LIN {X 0,Y 142.755,Z 442.404,A -85,B 0,C 180,E1 -25401.516,E2 -25401.516} C_VEL
LIN {X 0,Y 145.368,Z 446.098,A -85,B 0,C 180,E1 -25404.454,E2 -25404.454} C_VEL
LIN {X 0,Y 146.59,Z 447.682,A -85,B 0,C 180,E1 -25405.67,E2 -25405.67} C_VEL
LIN {X 0,Y 149.941,Z 452.496,A -85,B 0,C 180,E1 -25408.714,E2 -25408.714} C_VEL
LIN {X 0,Y 154.159,Z 458.757,A -85,B 0,C 180,E1 -25412.023,E2 -25412.023} C_VEL
LIN {X 0,Y 159.816,Z 468.413,A -85,B 0,C 180,E1 -25415.888,E2 -25415.888} C_VEL
LIN {X 0,Y 164.555,Z 477.501,A -85,B 0,C 180,E1 -25418.752,E2 -25418.752} C_VEL
LIN {X 0,Y 166.086,Z 481.604,A -85,B 0,C 180,E1 -25419.683,E2 -25419.683} C_VEL
LIN {X 0,Y 164.265,Z 506.272,A -85,B 0,C 180,E1 -25420.566,E2 -25420.566} C_VEL
LIN {X 0,Y 162.83,Z 520.798,A -85,B 0,C 180,E1 -25421.21,E2 -25421.21} C_VEL
LIN {X 0,Y 160.572,Z 533.522,A -85,B 0,C 180,E1 -25422.156,E2 -25422.156} C_VEL
LIN {X 0,Y 157.451,Z 545.977,A -85,B 0,C 180,E1 -25423.503,E2 -25423.503} C_VEL
LIN {X 0,Y 153.61,Z 557.923,A -85,B 0,C 180,E1 -25425.297,E2 -25425.297} C_VEL
LIN {X 0,Y 149.443,Z 568.566,A -85,B 0,C 180,E1 -25427.467,E2 -25427.467} C_VEL
LIN {X 0,Y 144.921,Z 578.272,A -85,B 0,C 180,E1 -25430.017,E2 -25430.017} C_VEL
LIN {X 0,Y 140.325,Z 587.101,A -85,B 0,C 180,E1 -25433.058,E2 -25433.058} C_VEL
LIN {X 0,Y 135.399,Z 595.708,A -85,B 0,C 180,E1 -25436.975,E2 -25436.975} C_VEL
LIN {X 0,Y 130.908,Z 602.575,A -85,B 0,C 180,E1 -25441.107,E2 -25441.107} C_VEL
LIN {X 0,Y 127.086,Z 608.071,A -85,B 0,C 180,E1 -25445.496,E2 -25445.496} C_VEL
LIN {X 0,Y 124.064,Z 612.381,A -85,B 0,C 180,E1 -25450.13,E2 -25450.13} C_VEL
LIN {X 0,Y 122.493,Z 614.66,A -85,B 0,C 180,E1 -25453.33,E2 -25453.33} C_VEL
LIN {X 0,Y 121.249,Z 616.511,A -85,B 0,C 180,E1 -25456.594,E2 -25456.594} C_VEL
LIN {X 0,Y 119.695,Z 618.888,A -85,B 0,C 180,E1 -25463.257,E2 -25463.257} C_VEL
LIN {X 0,Y 119.432,Z 619.492,A -85,B 0,C 180,E1 -25466.627,E2 -25466.627} C_VEL
LIN {X 0,Y 119.363,Z 619.717,A -85,B 0,C 180,E1 -25470.001,E2 -25470.001} C_VEL
LIN {X 0,Y 119.432,Z 619.521,A -85,B 0,C 180,E1 -25473.374,E2 -25473.374} C_VEL
LIN {X 0,Y 120.282,Z 617.966,A -85,B 0,C 180,E1 -25480.096,E2 -25480.096} C_VEL
LIN {X 0,Y 121.248,Z 616.605,A -85,B 0,C 180,E1 -25483.407,E2 -25483.407} C_VEL
LIN {X 0,Y 123.198,Z 613.733,A -85,B 0,C 180,E1 -25488.286,E2 -25488.286} C_VEL
LIN {X 0,Y 125.927,Z 609.834,A -85,B 0,C 180,E1 -25492.997,E2 -25492.997} C_VEL
LIN {X 0,Y 129.499,Z 604.802,A -85,B 0,C 180,E1 -25497.472,E2 -25497.472} C_VEL
LIN {X 0,Y 133.743,Z 598.462,A -85,B 0,C 180,E1 -25501.702,E2 -25501.702} C_VEL
LIN {X 0,Y 138.629,Z 590.323,A -85,B 0,C 180,E1 -25505.792,E2 -25505.792} C_VEL
LIN {X 0,Y 143.855,Z 580.672,A -85,B 0,C 180,E1 -25509.429,E2 -25509.429} C_VEL
LIN {X 0,Y 148.825,Z 570.306,A -85,B 0,C 180,E1 -25512.295,E2 -25512.295} C_VEL
LIN {X 0,Y 153.562,Z 558.617,A -85,B 0,C 180,E1 -25514.722,E2 -25514.722} C_VEL
LIN {X 0,Y 157.416,Z 546.938,A -85,B 0,C 180,E1 -25516.511,E2 -25516.511} C_VEL
LIN {X 0,Y 160.499,Z 534.785,A -85,B 0,C 180,E1 -25517.875,E2 -25517.875} C_VEL
LIN {X 0,Y 162.887,Z 521.701,A -85,B 0,C 180,E1 -25518.886,E2 -25518.886} C_VEL
LIN {X 0,Y 164.354,Z 508.522,A -85,B 0,C 180,E1 -25519.478,E2 -25519.478} C_VEL
LIN {X 0,Y 166.258,Z 481.734,A -85,B 0,C 180,E1 -25520.466,E2 -25520.466} C_VEL
LIN {X 0,Y 163.546,Z 475.199,A -85,B 0,C 180,E1 -25522.094,E2 -25522.094} C_VEL
LIN {X 0,Y 157.916,Z 464.862,A -85,B 0,C 180,E1 -25525.626,E2 -25525.626} C_VEL
LIN {X 0,Y 153.26,Z 457.318,A -85,B 0,C 180,E1 -25528.943,E2 -25528.943} C_VEL
LIN {X 0,Y 150.164,Z 452.699,A -85,B 0,C 180,E1 -25531.427,E2 -25531.427} C_VEL
LIN {X 0,Y 148.136,Z 449.857,A -85,B 0,C 180,E1 -25533.211,E2 -25533.211} C_VEL
LIN {X 0,Y 145.853,Z 446.536,A -85,B 0,C 180,E1 -25535.443,E2 -25535.443} C_VEL
LIN {X 0,Y 143.064,Z 442.903,A -85,B 0,C 180,E1 -25538.519,E2 -25538.519} C_VEL
LIN {X 0,Y 142.419,Z 441.849,A -85,B 0,C 180,E1 -25539.341,E2 -25539.341} C_VEL
LIN {X 0,Y 139.755,Z 438.86,A -85,B 0,C 180,E1 -25543.004,E2 -25543.004} C_VEL
LIN {X 0,Y 138.689,Z 436.693,A -85,B 0,C 180,E1 -25544.947,E2 -25544.947} C_VEL
LIN {X 0,Y 136.112,Z 434.575,A -85,B 0,C 180,E1 -25550.443,E2 -25550.443} C_VEL
LIN {X 0,Y 134.812,Z 430.977,A -85,B 0,C 180,E1 -25557.759,E2 -25557.759} C_VEL
LIN {X 0,Y 134.829,Z 431.049,A -85,B 0,C 180,E1 -25562.24,E2 -25562.24} C_VEL
LIN {X 0,Y 136.408,Z 435,A -85,B 0,C 180,E1 -25570.115,E2 -25570.115} C_VEL
LIN {X 0,Y 138.83,Z 436.963,A -85,B 0,C 180,E1 -25575.037,E2 -25575.037} C_VEL
LIN {X 0,Y 140.813,Z 440.378,A -85,B 0,C 180,E1 -25578.317,E2 -25578.317} C_VEL
LIN {X 0,Y 142.785,Z 442.377,A -85,B 0,C 180,E1 -25580.834,E2 -25580.834} C_VEL
LIN {X 0,Y 145.368,Z 446.062,A -85,B 0,C 180,E1 -25583.79,E2 -25583.79} C_VEL
LIN {X 0,Y 146.728,Z 447.809,A -85,B 0,C 180,E1 -25585.157,E2 -25585.157} C_VEL
LIN {X 0,Y 149.715,Z 452.036,A -85,B 0,C 180,E1 -25587.902,E2 -25587.902} C_VEL
LIN {X 0,Y 153.448,Z 457.658,A -85,B 0,C 180,E1 -25590.919,E2 -25590.919} C_VEL
LIN {X 0,Y 157.583,Z 465.906,A -85,B 0,C 180,E1 -25593.993,E2 -25593.993} C_VEL
LIN {X 0,Y 162.261,Z 476.642,A -85,B 0,C 180,E1 -25597.133,E2 -25597.133} C_VEL
LIN {X 0,Y 165.939,Z 486.652,A -85,B 0,C 180,E1 -25599.442,E2 -25599.442} C_VEL
LIN {X 0,Y 163.151,Z 522.008,A -85,B 0,C 180,E1 -25600.76,E2 -25600.76} C_VEL
LIN {X 0,Y 161.042,Z 535.203,A -85,B 0,C 180,E1 -25601.599,E2 -25601.599} C_VEL
LIN {X 0,Y 158.009,Z 547.842,A -85,B 0,C 180,E1 -25602.785,E2 -25602.785} C_VEL
LIN {X 0,Y 153.975,Z 560.493,A -85,B 0,C 180,E1 -25604.504,E2 -25604.504} C_VEL
LIN {X 0,Y 149.549,Z 571.749,A -85,B 0,C 180,E1 -25606.583,E2 -25606.583} C_VEL
LIN {X 0,Y 144.902,Z 581.889,A -85,B 0,C 180,E1 -25609.097,E2 -25609.097} C_VEL
LIN {X 0,Y 140.057,Z 591.027,A -85,B 0,C 180,E1 -25612.069,E2 -25612.069} C_VEL
LIN {X 0,Y 134.86,Z 599.939,A -85,B 0,C 180,E1 -25615.928,E2 -25615.928} C_VEL
LIN {X 0,Y 130.566,Z 607.116,A -85,B 0,C 180,E1 -25620.138,E2 -25620.138} C_VEL
LIN {X 0,Y 127.212,Z 611.956,A -85,B 0,C 180,E1 -25623.769,E2 -25623.769} C_VEL
LIN {X 0,Y 123.988,Z 616.664,A -85,B 0,C 180,E1 -25628.38,E2 -25628.38} C_VEL
LIN {X 0,Y 121.661,Z 620.264,A -85,B 0,C 180,E1 -25633.211,E2 -25633.211} C_VEL
LIN {X 0,Y 120.546,Z 622.121,A -85,B 0,C 180,E1 -25636.513,E2 -25636.513} C_VEL
LIN {X 0,Y 119.79,Z 623.516,A -85,B 0,C 180,E1 -25639.862,E2 -25639.862} C_VEL
LIN {X 0,Y 119.219,Z 625.123,A -85,B 0,C 180,E1 -25646.62,E2 -25646.62} C_VEL
LIN {X 0,Y 119.291,Z 625.336,A -85,B 0,C 180,E1 -25649.999,E2 -25649.999} C_VEL
LIN {X 0,Y 119.219,Z 625.107,A -85,B 0,C 180,E1 -25653.379,E2 -25653.379} C_VEL
LIN {X 0,Y 119.79,Z 623.48,A -85,B 0,C 180,E1 -25660.137,E2 -25660.137} C_VEL
LIN {X 0,Y 120.545,Z 622.069,A -85,B 0,C 180,E1 -25663.485,E2 -25663.485} C_VEL
LIN {X 0,Y 122.294,Z 619.116,A -85,B 0,C 180,E1 -25668.425,E2 -25668.425} C_VEL
LIN {X 0,Y 124.988,Z 615.13,A -85,B 0,C 180,E1 -25673.179,E2 -25673.179} C_VEL
LIN {X 0,Y 129.134,Z 609.004,A -85,B 0,C 180,E1 -25678.438,E2 -25678.438} C_VEL
LIN {X 0,Y 130.067,Z 607.646,A -85,B 0,C 180,E1 -25679.386,E2 -25679.386} C_VEL
LIN {X 0,Y 131.42,Z 604.603,A -85,B 0,C 180,E1 -25681.509,E2 -25681.509} C_VEL
LIN {X 0,Y 132.265,Z 599.24,A -85,B 0,C 180,E1 -25685.124,E2 -25685.124} C_VEL
LIN {X 0,Y 133.435,Z 593.402,A -85,B 0,C 180,E1 -25688.527,E2 -25688.527} C_VEL
LIN {X 0,Y 135.212,Z 589.419,A -85,B 0,C 180,E1 -25690.241,E2 -25690.241} C_VEL
LIN {X 0,Y 140.119,Z 580.38,A -85,B 0,C 180,E1 -25693.109,E2 -25693.109} C_VEL
LIN {X 0,Y 145.017,Z 569.915,A -85,B 0,C 180,E1 -25695.629,E2 -25695.629} C_VEL
LIN {X 0,Y 149.67,Z 558.285,A -85,B 0,C 180,E1 -25697.694,E2 -25697.694} C_VEL
LIN {X 0,Y 153.558,Z 545.907,A -85,B 0,C 180,E1 -25699.29,E2 -25699.29} C_VEL
LIN {X 0,Y 156.637,Z 533.099,A -85,B 0,C 180,E1 -25700.42,E2 -25700.42} C_VEL
LIN {X 0,Y 158.605,Z 520.451,A -85,B 0,C 180,E1 -25701.186,E2 -25701.186} C_VEL
LIN {X 0,Y 161.139,Z 488.74,A -85,B 0,C 180,E1 -25702.367,E2 -25702.367} C_VEL
LIN {X 0,Y 157.849,Z 479.526,A -85,B 0,C 180,E1 -25704.633,E2 -25704.633} C_VEL
LIN {X 0,Y 153.685,Z 469.729,A -85,B 0,C 180,E1 -25707.692,E2 -25707.692} C_VEL
LIN {X 0,Y 149.985,Z 462.282,A -85,B 0,C 180,E1 -25710.686,E2 -25710.686} C_VEL
LIN {X 0,Y 146.01,Z 456.208,A -85,B 0,C 180,E1 -25714.233,E2 -25714.233} C_VEL
LIN {X 0,Y 143.564,Z 452.633,A -85,B 0,C 180,E1 -25716.753,E2 -25716.753} C_VEL
LIN {X 0,Y 140.507,Z 448.264,A -85,B 0,C 180,E1 -25720.458,E2 -25720.458} C_VEL
LIN {X 0,Y 137.912,Z 444.918,A -85,B 0,C 180,E1 -25724.34,E2 -25724.34} C_VEL
LIN {X 0,Y 137.29,Z 443.587,A -85,B 0,C 180,E1 -25725.549,E2 -25725.549} C_VEL
LIN {X 0,Y 134.72,Z 441.175,A -85,B 0,C 180,E1 -25731.374,E2 -25731.374} C_VEL
LIN {X 0,Y 133.725,Z 438.021,A -85,B 0,C 180,E1 -25736.988,E2 -25736.988} C_VEL
LIN {X 0,Y 133.683,Z 437.987,A -85,B 0,C 180,E1 -25743.014,E2 -25743.014} C_VEL
LIN {X 0,Y 134.006,Z 439.323,A -85,B 0,C 180,E1 -25745.832,E2 -25745.832} C_VEL
LIN {X 0,Y 136.319,Z 442.986,A -85,B 0,C 180,E1 -25753.036,E2 -25753.036} C_VEL
LIN {X 0,Y 137.432,Z 443.82,A -85,B 0,C 180,E1 -25755.099,E2 -25755.099} C_VEL
LIN {X 0,Y 139.479,Z 447.275,A -85,B 0,C 180,E1 -25758.547,E2 -25758.547} C_VEL
LIN {X 0,Y 141.057,Z 449.016,A -85,B 0,C 180,E1 -25760.64,E2 -25760.64} C_VEL
LIN {X 0,Y 143.726,Z 452.8,A -85,B 0,C 180,E1 -25763.792,E2 -25763.792} C_VEL
LIN {X 0,Y 147.563,Z 458.511,A -85,B 0,C 180,E1 -25767.595,E2 -25767.595} C_VEL
LIN {X 0,Y 151.387,Z 464.47,A -85,B 0,C 180,E1 -25770.815,E2 -25770.815} C_VEL
LIN {X 0,Y 156.65,Z 473.786,A -85,B 0,C 180,E1 -25774.672,E2 -25774.672} C_VEL
LIN {X 0,Y 160.86,Z 482.253,A -85,B 0,C 180,E1 -25777.415,E2 -25777.415} C_VEL
LIN {X 0,Y 161.489,Z 484.052,A -85,B 0,C 180,E1 -25777.836,E2 -25777.836} C_VEL
LIN {X 0,Y 159.701,Z 506.929,A -85,B 0,C 180,E1 -25778.647,E2 -25778.647} C_VEL
LIN {X 0,Y 158.217,Z 521.237,A -85,B 0,C 180,E1 -25779.296,E2 -25779.296} C_VEL
LIN {X 0,Y 155.911,Z 533.697,A -85,B 0,C 180,E1 -25780.227,E2 -25780.227} C_VEL
LIN {X 0,Y 152.661,Z 546.15,A -85,B 0,C 180,E1 -25781.575,E2 -25781.575} C_VEL
LIN {X 0,Y 148.664,Z 558.094,A -85,B 0,C 180,E1 -25783.378,E2 -25783.378} C_VEL
LIN {X 0,Y 144.295,Z 568.737,A -85,B 0,C 180,E1 -25785.562,E2 -25785.562} C_VEL
LIN {X 0,Y 139.546,Z 578.443,A -85,B 0,C 180,E1 -25788.14,E2 -25788.14} C_VEL
LIN {X 0,Y 134.707,Z 587.271,A -85,B 0,C 180,E1 -25791.24,E2 -25791.24} C_VEL
LIN {X 0,Y 129.479,Z 595.878,A -85,B 0,C 180,E1 -25795.255,E2 -25795.255} C_VEL
LIN {X 0,Y 124.737,Z 602.744,A -85,B 0,C 180,E1 -25799.531,E2 -25799.531} C_VEL
LIN {X 0,Y 120.653,Z 608.24,A -85,B 0,C 180,E1 -25804.096,E2 -25804.096} C_VEL
LIN {X 0,Y 117.411,Z 612.55,A -85,B 0,C 180,E1 -25808.953,E2 -25808.953} C_VEL
LIN {X 0,Y 115.688,Z 614.829,A -85,B 0,C 180,E1 -25812.318,E2 -25812.318} C_VEL
LIN {X 0,Y 114.357,Z 616.679,A -85,B 0,C 180,E1 -25815.77,E2 -25815.77} C_VEL
LIN {X 0,Y 112.637,Z 619.056,A -85,B 0,C 180,E1 -25822.832,E2 -25822.832} C_VEL
LIN {X 0,Y 112.351,Z 619.659,A -85,B 0,C 180,E1 -25826.414,E2 -25826.414} C_VEL
LIN {X 0,Y 112.266,Z 619.884,A -85,B 0,C 180,E1 -25830.001,E2 -25830.001} C_VEL
LIN {X 0,Y 112.351,Z 619.688,A -85,B 0,C 180,E1 -25833.587,E2 -25833.587} C_VEL
LIN {X 0,Y 113.305,Z 618.133,A -85,B 0,C 180,E1 -25840.725,E2 -25840.725} C_VEL
LIN {X 0,Y 114.356,Z 616.772,A -85,B 0,C 180,E1 -25844.232,E2 -25844.232} C_VEL
LIN {X 0,Y 116.477,Z 613.899,A -85,B 0,C 180,E1 -25849.382,E2 -25849.382} C_VEL
LIN {X 0,Y 119.403,Z 610.001,A -85,B 0,C 180,E1 -25854.332,E2 -25854.332} C_VEL
LIN {X 0,Y 123.251,Z 604.967,A -85,B 0,C 180,E1 -25858.993,E2 -25858.993} C_VEL
LIN {X 0,Y 127.747,Z 598.627,A -85,B 0,C 180,E1 -25863.378,E2 -25863.378} C_VEL
LIN {X 0,Y 132.56,Z 591.086,A -85,B 0,C 180,E1 -25867.319,E2 -25867.319} C_VEL
LIN {X 0,Y 137.451,Z 582.616,A -85,B 0,C 180,E1 -25870.688,E2 -25870.688} C_VEL
LIN {X 0,Y 142.579,Z 572.747,A -85,B 0,C 180,E1 -25873.638,E2 -25873.638} C_VEL
LIN {X 0,Y 147.482,Z 561.626,A -85,B 0,C 180,E1 -25876.118,E2 -25876.118} C_VEL
LIN {X 0,Y 151.445,Z 550.723,A -85,B 0,C 180,E1 -25877.946,E2 -25877.946} C_VEL
LIN {X 0,Y 154.953,Z 538.665,A -85,B 0,C 180,E1 -25879.44,E2 -25879.44} C_VEL
LIN {X 0,Y 157.677,Z 525.917,A -85,B 0,C 180,E1 -25880.544,E2 -25880.544} C_VEL
LIN {X 0,Y 159.479,Z 512.518,A -85,B 0,C 180,E1 -25881.269,E2 -25881.269} C_VEL
LIN {X 0,Y 161.696,Z 484.326,A -85,B 0,C 180,E1 -25882.292,E2 -25882.292} C_VEL
LIN {X 0,Y 159.447,Z 478.95,A -85,B 0,C 180,E1 -25883.757,E2 -25883.757} C_VEL
LIN {X 0,Y 154.315,Z 469.367,A -85,B 0,C 180,E1 -25887.26,E2 -25887.26} C_VEL
LIN {X 0,Y 149.91,Z 461.957,A -85,B 0,C 180,E1 -25890.702,E2 -25890.702} C_VEL
LIN {X 0,Y 146.165,Z 456.308,A -85,B 0,C 180,E1 -25894.071,E2 -25894.071} C_VEL
LIN {X 0,Y 143.734,Z 452.767,A -85,B 0,C 180,E1 -25896.592,E2 -25896.592} C_VEL
LIN {X 0,Y 140.57,Z 448.282,A -85,B 0,C 180,E1 -25900.467,E2 -25900.467} C_VEL
LIN {X 0,Y 138.049,Z 445.022,A -85,B 0,C 180,E1 -25904.308,E2 -25904.308} C_VEL
LIN {X 0,Y 137.323,Z 443.56,A -85,B 0,C 180,E1 -25905.741,E2 -25905.741} C_VEL
LIN {X 0,Y 134.628,Z 440.76,A -85,B 0,C 180,E1 -25912.502,E2 -25912.502} C_VEL
LIN {X 0,Y 133.939,Z 438.086,A -85,B 0,C 180,E1 -25917.744,E2 -25917.744} C_VEL
LIN {X 0,Y 133.942,Z 438.131,A -85,B 0,C 180,E1 -25922.067,E2 -25922.067} C_VEL
LIN {X 0,Y 135.244,Z 441.819,A -85,B 0,C 180,E1 -25929.354,E2 -25929.354} C_VEL
LIN {X 0,Y 137.505,Z 443.86,A -85,B 0,C 180,E1 -25934.334,E2 -25934.334} C_VEL
LIN {X 0,Y 139.495,Z 447.257,A -85,B 0,C 180,E1 -25937.784,E2 -25937.784} C_VEL
LIN {X 0,Y 141.119,Z 449,A -85,B 0,C 180,E1 -25939.976,E2 -25939.976} C_VEL
LIN {X 0,Y 143.762,Z 452.792,A -85,B 0,C 180,E1 -25943.152,E2 -25943.152} C_VEL
LIN {X 0,Y 147.394,Z 458.152,A -85,B 0,C 180,E1 -25946.809,E2 -25946.809} C_VEL
LIN {X 0,Y 150.857,Z 463.633,A -85,B 0,C 180,E1 -25949.807,E2 -25949.807} C_VEL
LIN {X 0,Y 154.954,Z 472.375,A -85,B 0,C 180,E1 -25953.071,E2 -25953.071} C_VEL
LIN {X 0,Y 159.283,Z 483.061,A -85,B 0,C 180,E1 -25956.184,E2 -25956.184} C_VEL
LIN {X 0,Y 161.326,Z 488.965,A -85,B 0,C 180,E1 -25957.582,E2 -25957.582} C_VEL
LIN {X 0,Y 158.621,Z 521.753,A -85,B 0,C 180,E1 -25958.812,E2 -25958.812} C_VEL
LIN {X 0,Y 156.347,Z 535.392,A -85,B 0,C 180,E1 -25959.679,E2 -25959.679} C_VEL
LIN {X 0,Y 153.286,Z 547.682,A -85,B 0,C 180,E1 -25960.842,E2 -25960.842} C_VEL
LIN {X 0,Y 149.09,Z 560.331,A -85,B 0,C 180,E1 -25962.56,E2 -25962.56} C_VEL
LIN {X 0,Y 144.47,Z 571.586,A -85,B 0,C 180,E1 -25964.645,E2 -25964.645} C_VEL
LIN {X 0,Y 139.595,Z 581.724,A -85,B 0,C 180,E1 -25967.181,E2 -25967.181} C_VEL
LIN {X 0,Y 134.523,Z 590.863,A -85,B 0,C 180,E1 -25970.208,E2 -25970.208} C_VEL
LIN {X 0,Y 129.004,Z 599.773,A -85,B 0,C 180,E1 -25974.15,E2 -25974.15} C_VEL
LIN {X 0,Y 124.632,Z 606.616,A -85,B 0,C 180,E1 -25978.271,E2 -25978.271} C_VEL
LIN {X 0,Y 120.849,Z 611.79,A -85,B 0,C 180,E1 -25982.273,E2 -25982.273} C_VEL
LIN {X 0,Y 117.402,Z 616.497,A -85,B 0,C 180,E1 -25987.1,E2 -25987.1} C_VEL
LIN {X 0,Y 114.828,Z 620.097,A -85,B 0,C 180,E1 -25992.18,E2 -25992.18} C_VEL
LIN {X 0,Y 113.638,Z 621.954,A -85,B 0,C 180,E1 -25995.677,E2 -25995.677} C_VEL
LIN {X 0,Y 112.783,Z 623.348,A -85,B 0,C 180,E1 -25999.225,E2 -25999.225} C_VEL
LIN {X 0,Y 112.127,Z 624.956,A -85,B 0,C 180,E1 -26006.406,E2 -26006.406} C_VEL
LIN {X 0,Y 112.204,Z 625.169,A -85,B 0,C 180,E1 -26009.999,E2 -26009.999} C_VEL
LIN {X 0,Y 112.127,Z 624.939,A -85,B 0,C 180,E1 -26013.593,E2 -26013.593} C_VEL
LIN {X 0,Y 112.782,Z 623.312,A -85,B 0,C 180,E1 -26020.774,E2 -26020.774} C_VEL
LIN {X 0,Y 113.637,Z 621.901,A -85,B 0,C 180,E1 -26024.322,E2 -26024.322} C_VEL
LIN {X 0,Y 115.542,Z 618.947,A -85,B 0,C 180,E1 -26029.544,E2 -26029.544} C_VEL
LIN {X 0,Y 118.477,Z 614.961,A -85,B 0,C 180,E1 -26034.534,E2 -26034.534} C_VEL
LIN {X 0,Y 122.939,Z 608.836,A -85,B 0,C 180,E1 -26040.013,E2 -26040.013} C_VEL
LIN {X 0,Y 127.337,Z 602.144,A -85,B 0,C 180,E1 -26044.452,E2 -26044.452} C_VEL
LIN {X 0,Y 132.589,Z 593.852,A -85,B 0,C 180,E1 -26048.522,E2 -26048.522} C_VEL
LIN {X 0,Y 135.212,Z 589.419,A -85,B 0,C 180,E1 -26050.241,E2 -26050.241} C_VEL
LIN {X 0,Y 137.042,Z 585.294,A -85,B 0,C 180,E1 -26051.854,E2 -26051.854} C_VEL
LIN {X 0,Y 138.616,Z 578.295,A -85,B 0,C 180,E1 -26054.712,E2 -26054.712} C_VEL
LIN {X 0,Y 140.164,Z 570.804,A -85,B 0,C 180,E1 -26057.301,E2 -26057.301} C_VEL
LIN {X 0,Y 141.856,Z 565.912,A -85,B 0,C 180,E1 -26058.452,E2 -26058.452} C_VEL
LIN {X 0,Y 146.193,Z 554.627,A -85,B 0,C 180,E1 -26060.28,E2 -26060.28} C_VEL
LIN {X 0,Y 149.712,Z 543.473,A -85,B 0,C 180,E1 -26061.57,E2 -26061.57} C_VEL
LIN {X 0,Y 152.608,Z 530.793,A -85,B 0,C 180,E1 -26062.652,E2 -26062.652} C_VEL
LIN {X 0,Y 154.612,Z 517.043,A -85,B 0,C 180,E1 -26063.362,E2 -26063.362} C_VEL
LIN {X 0,Y 156.694,Z 491.085,A -85,B 0,C 180,E1 -26064.333,E2 -26064.333} C_VEL
LIN {X 0,Y 153.873,Z 483.038,A -85,B 0,C 180,E1 -26066.47,E2 -26066.47} C_VEL
LIN {X 0,Y 150.323,Z 474.307,A -85,B 0,C 180,E1 -26069.343,E2 -26069.343} C_VEL
LIN {X 0,Y 147.322,Z 467.959,A -85,B 0,C 180,E1 -26071.992,E2 -26071.992} C_VEL
LIN {X 0,Y 143.587,Z 461.978,A -85,B 0,C 180,E1 -26075.608,E2 -26075.608} C_VEL
LIN {X 0,Y 141.598,Z 458.922,A -85,B 0,C 180,E1 -26077.827,E2 -26077.827} C_VEL
LIN {X 0,Y 138.937,Z 454.909,A -85,B 0,C 180,E1 -26081.283,E2 -26081.283} C_VEL
LIN {X 0,Y 136.459,Z 451.518,A -85,B 0,C 180,E1 -26085.268,E2 -26085.268} C_VEL
LIN {X 0,Y 135.952,Z 450.407,A -85,B 0,C 180,E1 -26086.332,E2 -26086.332} C_VEL
LIN {X 0,Y 133.534,Z 447.805,A -85,B 0,C 180,E1 -26092.439,E2 -26092.439} C_VEL
LIN {X 0,Y 132.78,Z 445.014,A -85,B 0,C 180,E1 -26097.725,E2 -26097.725} C_VEL
LIN {X 0,Y 132.815,Z 445.063,A -85,B 0,C 180,E1 -26103.033,E2 -26103.033} C_VEL
LIN {X 0,Y 135.169,Z 449.879,A -85,B 0,C 180,E1 -26112.5,E2 -26112.5} C_VEL
LIN {X 0,Y 136.117,Z 450.709,A -85,B 0,C 180,E1 -26114.388,E2 -26114.388} C_VEL
LIN {X 0,Y 138.377,Z 454.372,A -85,B 0,C 180,E1 -26118.316,E2 -26118.316} C_VEL
LIN {X 0,Y 139.49,Z 455.825,A -85,B 0,C 180,E1 -26119.883,E2 -26119.883} C_VEL
LIN {X 0,Y 142.679,Z 460.552,A -85,B 0,C 180,E1 -26123.785,E2 -26123.785} C_VEL
LIN {X 0,Y 145.645,Z 465.222,A -85,B 0,C 180,E1 -26126.835,E2 -26126.835} C_VEL
LIN {X 0,Y 148.954,Z 470.681,A -85,B 0,C 180,E1 -26129.795,E2 -26129.795} C_VEL
LIN {X 0,Y 153.617,Z 479.373,A -85,B 0,C 180,E1 -26133.458,E2 -26133.458} C_VEL
LIN {X 0,Y 157.043,Z 486.453,A -85,B 0,C 180,E1 -26135.865,E2 -26135.865} C_VEL
LIN {X 0,Y 155.473,Z 506.095,A -85,B 0,C 180,E1 -26136.577,E2 -26136.577} C_VEL
LIN {X 0,Y 153.871,Z 521.114,A -85,B 0,C 180,E1 -26137.235,E2 -26137.235} C_VEL
LIN {X 0,Y 151.431,Z 533.872,A -85,B 0,C 180,E1 -26138.18,E2 -26138.18} C_VEL
LIN {X 0,Y 148.056,Z 546.324,A -85,B 0,C 180,E1 -26139.524,E2 -26139.524} C_VEL
LIN {X 0,Y 143.899,Z 558.266,A -85,B 0,C 180,E1 -26141.331,E2 -26141.331} C_VEL
LIN {X 0,Y 139.324,Z 568.907,A -85,B 0,C 180,E1 -26143.521,E2 -26143.521} C_VEL
LIN {X 0,Y 134.343,Z 578.613,A -85,B 0,C 180,E1 -26146.12,E2 -26146.12} C_VEL
LIN {X 0,Y 129.234,Z 587.441,A -85,B 0,C 180,E1 -26149.264,E2 -26149.264} C_VEL
LIN {X 0,Y 123.684,Z 596.048,A -85,B 0,C 180,E1 -26153.371,E2 -26153.371} C_VEL
LIN {X 0,Y 118.673,Z 602.912,A -85,B 0,C 180,E1 -26157.793,E2 -26157.793} C_VEL
LIN {X 0,Y 114.308,Z 608.409,A -85,B 0,C 180,E1 -26162.541,E2 -26162.541} C_VEL
LIN {X 0,Y 110.818,Z 612.718,A -85,B 0,C 180,E1 -26167.635,E2 -26167.635} C_VEL
LIN {X 0,Y 108.936,Z 614.997,A -85,B 0,C 180,E1 -26171.182,E2 -26171.182} C_VEL
LIN {X 0,Y 107.476,Z 616.847,A -85,B 0,C 180,E1 -26174.838,E2 -26174.838} C_VEL
LIN {X 0,Y 105.608,Z 619.223,A -85,B 0,C 180,E1 -26182.352,E2 -26182.352} C_VEL
LIN {X 0,Y 105.264,Z 619.827,A -85,B 0,C 180,E1 -26186.172,E2 -26186.172} C_VEL
LIN {X 0,Y 105.18,Z 620.051,A -85,B 0,C 180,E1 -26190.001,E2 -26190.001} C_VEL
LIN {X 0,Y 105.265,Z 619.855,A -85,B 0,C 180,E1 -26193.829,E2 -26193.829} C_VEL
LIN {X 0,Y 106.333,Z 618.3,A -85,B 0,C 180,E1 -26201.437,E2 -26201.437} C_VEL
LIN {X 0,Y 107.474,Z 616.939,A -85,B 0,C 180,E1 -26205.164,E2 -26205.164} C_VEL
LIN {X 0,Y 109.81,Z 614.065,A -85,B 0,C 180,E1 -26210.611,E2 -26210.611} C_VEL
LIN {X 0,Y 112.954,Z 610.167,A -85,B 0,C 180,E1 -26215.821,E2 -26215.821} C_VEL
LIN {X 0,Y 117.101,Z 605.133,A -85,B 0,C 180,E1 -26220.674,E2 -26220.674} C_VEL
LIN {X 0,Y 121.869,Z 598.793,A -85,B 0,C 180,E1 -26225.219,E2 -26225.219} C_VEL
LIN {X 0,Y 127.355,Z 590.659,A -85,B 0,C 180,E1 -26229.535,E2 -26229.535} C_VEL
LIN {X 0,Y 133.183,Z 581.001,A -85,B 0,C 180,E1 -26233.316,E2 -26233.316} C_VEL
LIN {X 0,Y 138.661,Z 570.632,A -85,B 0,C 180,E1 -26236.242,E2 -26236.242} C_VEL
LIN {X 0,Y 143.242,Z 560.365,A -85,B 0,C 180,E1 -26238.438,E2 -26238.438} C_VEL
LIN {X 0,Y 147.415,Z 549.122,A -85,B 0,C 180,E1 -26240.244,E2 -26240.244} C_VEL
LIN {X 0,Y 150.75,Z 537.679,A -85,B 0,C 180,E1 -26241.611,E2 -26241.611} C_VEL
LIN {X 0,Y 153.547,Z 524.396,A -85,B 0,C 180,E1 -26242.703,E2 -26242.703} C_VEL
LIN {X 0,Y 155.346,Z 510.753,A -85,B 0,C 180,E1 -26243.383,E2 -26243.383} C_VEL
LIN {X 0,Y 157.256,Z 486.735,A -85,B 0,C 180,E1 -26244.264,E2 -26244.264} C_VEL
LIN {X 0,Y 153.166,Z 478.211,A -85,B 0,C 180,E1 -26247.179,E2 -26247.179} C_VEL
LIN {X 0,Y 148.541,Z 469.747,A -85,B 0,C 180,E1 -26250.892,E2 -26250.892} C_VEL
LIN {X 0,Y 144.553,Z 463.18,A -85,B 0,C 180,E1 -26254.63,E2 -26254.63} C_VEL
LIN {X 0,Y 141.678,Z 458.94,A -85,B 0,C 180,E1 -26257.777,E2 -26257.777} C_VEL
LIN {X 0,Y 138.947,Z 454.896,A -85,B 0,C 180,E1 -26261.38,E2 -26261.38} C_VEL
LIN {X 0,Y 136.5,Z 451.384,A -85,B 0,C 180,E1 -26265.463,E2 -26265.463} C_VEL
LIN {X 0,Y 135.988,Z 450.385,A -85,B 0,C 180,E1 -26266.552,E2 -26266.552} C_VEL
LIN {X 0,Y 133.158,Z 446.378,A -85,B 0,C 180,E1 -26275.838,E2 -26275.838} C_VEL
LIN {X 0,Y 133.033,Z 445.034,A -85,B 0,C 180,E1 -26278.486,E2 -26278.486} C_VEL
LIN {X 0,Y 133.04,Z 445.235,A -85,B 0,C 180,E1 -26281.703,E2 -26281.703} C_VEL
LIN {X 0,Y 135.077,Z 449.758,A -85,B 0,C 180,E1 -26291.251,E2 -26291.251} C_VEL
LIN {X 0,Y 136.243,Z 450.844,A -85,B 0,C 180,E1 -26293.707,E2 -26293.707} C_VEL
LIN {X 0,Y 138.28,Z 454.211,A -85,B 0,C 180,E1 -26297.373,E2 -26297.373} C_VEL
LIN {X 0,Y 139.493,Z 455.693,A -85,B 0,C 180,E1 -26299.116,E2 -26299.116} C_VEL
LIN {X 0,Y 142.767,Z 460.558,A -85,B 0,C 180,E1 -26303.192,E2 -26303.192} C_VEL
LIN {X 0,Y 145.67,Z 465.156,A -85,B 0,C 180,E1 -26306.216,E2 -26306.216} C_VEL
LIN {X 0,Y 148.259,Z 469.504,A -85,B 0,C 180,E1 -26308.6,E2 -26308.6} C_VEL
LIN {X 0,Y 151.938,Z 477.824,A -85,B 0,C 180,E1 -26311.773,E2 -26311.773} C_VEL
LIN {X 0,Y 155.723,Z 487.762,A -85,B 0,C 180,E1 -26314.736,E2 -26314.736} C_VEL
LIN {X 0,Y 156.893,Z 491.273,A -85,B 0,C 180,E1 -26315.615,E2 -26315.615} C_VEL
LIN {X 0,Y 154.294,Z 521.354,A -85,B 0,C 180,E1 -26316.739,E2 -26316.739} C_VEL
LIN {X 0,Y 151.952,Z 535.052,A -85,B 0,C 180,E1 -26317.605,E2 -26317.605} C_VEL
LIN {X 0,Y 148.751,Z 547.522,A -85,B 0,C 180,E1 -26318.777,E2 -26318.777} C_VEL
LIN {X 0,Y 144.39,Z 560.169,A -85,B 0,C 180,E1 -26320.488,E2 -26320.488} C_VEL
LIN {X 0,Y 139.563,Z 571.423,A -85,B 0,C 180,E1 -26322.567,E2 -26322.567} C_VEL
LIN {X 0,Y 134.467,Z 581.56,A -85,B 0,C 180,E1 -26325.122,E2 -26325.122} C_VEL
LIN {X 0,Y 129.143,Z 590.698,A -85,B 0,C 180,E1 -26328.19,E2 -26328.19} C_VEL
LIN {X 0,Y 123.302,Z 599.608,A -85,B 0,C 180,E1 -26332.212,E2 -26332.212} C_VEL
LIN {X 0,Y 118.44,Z 606.703,A -85,B 0,C 180,E1 -26336.634,E2 -26336.634} C_VEL
LIN {X 0,Y 114.588,Z 611.623,A -85,B 0,C 180,E1 -26340.615,E2 -26340.615} C_VEL
LIN {X 0,Y 110.885,Z 616.331,A -85,B 0,C 180,E1 -26345.67,E2 -26345.67} C_VEL
LIN {X 0,Y 108.042,Z 619.929,A -85,B 0,C 180,E1 -26351.019,E2 -26351.019} C_VEL
LIN {X 0,Y 106.746,Z 621.787,A -85,B 0,C 180,E1 -26354.73,E2 -26354.73} C_VEL
LIN {X 0,Y 105.804,Z 623.181,A -85,B 0,C 180,E1 -26358.505,E2 -26358.505} C_VEL
LIN {X 0,Y 105.035,Z 624.789,A -85,B 0,C 180,E1 -26366.163,E2 -26366.163} C_VEL
LIN {X 0,Y 105.108,Z 625.002,A -85,B 0,C 180,E1 -26369.999,E2 -26369.999} C_VEL
LIN {X 0,Y 105.035,Z 624.772,A -85,B 0,C 180,E1 -26373.836,E2 -26373.836} C_VEL
LIN {X 0,Y 105.803,Z 623.144,A -85,B 0,C 180,E1 -26381.494,E2 -26381.494} C_VEL
LIN {X 0,Y 106.745,Z 621.732,A -85,B 0,C 180,E1 -26385.269,E2 -26385.269} C_VEL
LIN {X 0,Y 108.849,Z 618.778,A -85,B 0,C 180,E1 -26390.8,E2 -26390.8} C_VEL
LIN {X 0,Y 112.043,Z 614.793,A -85,B 0,C 180,E1 -26396.045,E2 -26396.045} C_VEL
LIN {X 0,Y 116.842,Z 608.667,A -85,B 0,C 180,E1 -26401.756,E2 -26401.756} C_VEL
LIN {X 0,Y 121.515,Z 601.974,A -85,B 0,C 180,E1 -26406.357,E2 -26406.357} C_VEL
LIN {X 0,Y 127.103,Z 593.682,A -85,B 0,C 180,E1 -26410.519,E2 -26410.519} C_VEL
LIN {X 0,Y 132.26,Z 585.176,A -85,B 0,C 180,E1 -26413.692,E2 -26413.692} C_VEL
LIN {X 0,Y 137.836,Z 574.669,A -85,B 0,C 180,E1 -26416.6,E2 -26416.6} C_VEL
LIN {X 0,Y 141.856,Z 565.912,A -85,B 0,C 180,E1 -26418.452,E2 -26418.452} C_VEL
LIN {X 0,Y 142.807,Z 562.571,A -85,B 0,C 180,E1 -26419.26,E2 -26419.26} C_VEL
LIN {X 0,Y 143.008,Z 551.955,A -85,B 0,C 180,E1 -26422.641,E2 -26422.641} C_VEL
LIN {X 0,Y 143.812,Z 548.399,A -85,B 0,C 180,E1 -26423.252,E2 -26423.252} C_VEL
LIN {X 0,Y 147.071,Z 537.003,A -85,B 0,C 180,E1 -26424.327,E2 -26424.327} C_VEL
LIN {X 0,Y 149.587,Z 523.871,A -85,B 0,C 180,E1 -26425.217,E2 -26425.217} C_VEL
LIN {X 0,Y 151.286,Z 507.73,A -85,B 0,C 180,E1 -26425.874,E2 -26425.874} C_VEL
LIN {X 0,Y 152.439,Z 493.48,A -85,B 0,C 180,E1 -26426.41,E2 -26426.41} C_VEL
LIN {X 0,Y 149.359,Z 484.522,A -85,B 0,C 180,E1 -26429.025,E2 -26429.025} C_VEL
LIN {X 0,Y 146.002,Z 476.31,A -85,B 0,C 180,E1 -26432.107,E2 -26432.107} C_VEL
LIN {X 0,Y 144.12,Z 472.445,A -85,B 0,C 180,E1 -26433.967,E2 -26433.967} C_VEL
LIN {X 0,Y 140.101,Z 465.762,A -85,B 0,C 180,E1 -26438.42,E2 -26438.42} C_VEL
LIN {X 0,Y 137.177,Z 461.352,A -85,B 0,C 180,E1 -26442.444,E2 -26442.444} C_VEL
LIN {X 0,Y 134.85,Z 457.647,A -85,B 0,C 180,E1 -26446.656,E2 -26446.656} C_VEL
LIN {X 0,Y 134.09,Z 456.84,A -85,B 0,C 180,E1 -26448.282,E2 -26448.282} C_VEL
LIN {X 0,Y 132,Z 452.997,A -85,B 0,C 180,E1 -26456.184,E2 -26456.184} C_VEL
LIN {X 0,Y 131.908,Z 452.126,A -85,B 0,C 180,E1 -26457.71,E2 -26457.71} C_VEL
LIN {X 0,Y 131.913,Z 452.088,A -85,B 0,C 180,E1 -26462.672,E2 -26462.672} C_VEL
LIN {X 0,Y 133.945,Z 456.674,A -85,B 0,C 180,E1 -26471.752,E2 -26471.752} C_VEL
LIN {X 0,Y 134.867,Z 457.662,A -85,B 0,C 180,E1 -26473.754,E2 -26473.754} C_VEL
LIN {X 0,Y 137.278,Z 461.468,A -85,B 0,C 180,E1 -26478.082,E2 -26478.082} C_VEL
LIN {X 0,Y 140.674,Z 466.819,A -85,B 0,C 180,E1 -26482.673,E2 -26482.673} C_VEL
LIN {X 0,Y 143.804,Z 471.93,A -85,B 0,C 180,E1 -26486.095,E2 -26486.095} C_VEL
LIN {X 0,Y 147.643,Z 478.908,A -85,B 0,C 180,E1 -26489.693,E2 -26489.693} C_VEL
LIN {X 0,Y 151.975,Z 487.663,A -85,B 0,C 180,E1 -26493.213,E2 -26493.213} C_VEL
LIN {X 0,Y 152.743,Z 489.3,A -85,B 0,C 180,E1 -26493.79,E2 -26493.79} C_VEL
LIN {X 0,Y 151.44,Z 505.399,A -85,B 0,C 180,E1 -26494.395,E2 -26494.395} C_VEL
LIN {X 0,Y 149.814,Z 520.494,A -85,B 0,C 180,E1 -26495.038,E2 -26495.038} C_VEL
LIN {X 0,Y 147.464,Z 532.745,A -85,B 0,C 180,E1 -26495.885,E2 -26495.885} C_VEL
LIN {X 0,Y 144.276,Z 544.512,A -85,B 0,C 180,E1 -26497.093,E2 -26497.093} C_VEL
LIN {X 0,Y 140.579,Z 555.296,A -85,B 0,C 180,E1 -26498.635,E2 -26498.635} C_VEL
LIN {X 0,Y 135.687,Z 566.624,A -85,B 0,C 180,E1 -26500.755,E2 -26500.755} C_VEL
LIN {X 0,Y 130.44,Z 576.83,A -85,B 0,C 180,E1 -26503.334,E2 -26503.334} C_VEL
LIN {X 0,Y 124.954,Z 585.991,A -85,B 0,C 180,E1 -26506.45,E2 -26506.45} C_VEL
LIN {X 0,Y 119.002,Z 594.891,A -85,B 0,C 180,E1 -26510.59,E2 -26510.59} C_VEL
LIN {X 0,Y 113.594,Z 602.056,A -85,B 0,C 180,E1 -26515.09,E2 -26515.09} C_VEL
LIN {X 0,Y 109.513,Z 606.887,A -85,B 0,C 180,E1 -26519.11,E2 -26519.11} C_VEL
LIN {X 0,Y 105.445,Z 611.578,A -85,B 0,C 180,E1 -26524.328,E2 -26524.328} C_VEL
LIN {X 0,Y 102.241,Z 615.165,A -85,B 0,C 180,E1 -26529.898,E2 -26529.898} C_VEL
LIN {X 0,Y 100.637,Z 617.015,A -85,B 0,C 180,E1 -26533.78,E2 -26533.78} C_VEL
LIN {X 0,Y 98.571,Z 619.39,A -85,B 0,C 180,E1 -26541.803,E2 -26541.803} C_VEL
LIN {X 0,Y 98.189,Z 619.994,A -85,B 0,C 180,E1 -26545.896,E2 -26545.896} C_VEL
LIN {X 0,Y 98.086,Z 620.218,A -85,B 0,C 180,E1 -26550.001,E2 -26550.001} C_VEL
LIN {X 0,Y 98.189,Z 620.021,A -85,B 0,C 180,E1 -26554.105,E2 -26554.105} C_VEL
LIN {X 0,Y 99.373,Z 618.467,A -85,B 0,C 180,E1 -26562.25,E2 -26562.25} C_VEL
LIN {X 0,Y 100.635,Z 617.105,A -85,B 0,C 180,E1 -26566.222,E2 -26566.222} C_VEL
LIN {X 0,Y 103.184,Z 614.232,A -85,B 0,C 180,E1 -26572.001,E2 -26572.001} C_VEL
LIN {X 0,Y 106.594,Z 610.334,A -85,B 0,C 180,E1 -26577.487,E2 -26577.487} C_VEL
LIN {X 0,Y 111.051,Z 605.299,A -85,B 0,C 180,E1 -26582.544,E2 -26582.544} C_VEL
LIN {X 0,Y 116.125,Z 598.958,A -85,B 0,C 180,E1 -26587.245,E2 -26587.245} C_VEL
LIN {X 0,Y 121.624,Z 591.325,A -85,B 0,C 180,E1 -26591.426,E2 -26591.426} C_VEL
LIN {X 0,Y 127.021,Z 582.944,A -85,B 0,C 180,E1 -26594.867,E2 -26594.867} C_VEL
LIN {X 0,Y 132.693,Z 573.073,A -85,B 0,C 180,E1 -26597.861,E2 -26597.861} C_VEL
LIN {X 0,Y 138.021,Z 561.951,A -85,B 0,C 180,E1 -26600.37,E2 -26600.37} C_VEL
LIN {X 0,Y 142.326,Z 551.046,A -85,B 0,C 180,E1 -26602.193,E2 -26602.193} C_VEL
LIN {X 0,Y 146.133,Z 538.984,A -85,B 0,C 180,E1 -26603.666,E2 -26603.666} C_VEL
LIN {X 0,Y 149.075,Z 526.105,A -85,B 0,C 180,E1 -26604.772,E2 -26604.772} C_VEL
LIN {X 0,Y 150.97,Z 513.245,A -85,B 0,C 180,E1 -26605.451,E2 -26605.451} C_VEL
LIN {X 0,Y 152.986,Z 489.53,A -85,B 0,C 180,E1 -26606.329,E2 -26606.329} C_VEL
LIN {X 0,Y 148.49,Z 480.275,A -85,B 0,C 180,E1 -26609.913,E2 -26609.913} C_VEL
LIN {X 0,Y 144.531,Z 472.893,A -85,B 0,C 180,E1 -26613.561,E2 -26613.561} C_VEL
LIN {X 0,Y 140.379,Z 466.037,A -85,B 0,C 180,E1 -26618.142,E2 -26618.142} C_VEL
LIN {X 0,Y 137.248,Z 461.345,A -85,B 0,C 180,E1 -26622.492,E2 -26622.492} C_VEL
LIN {X 0,Y 135.009,Z 457.741,A -85,B 0,C 180,E1 -26626.644,E2 -26626.644} C_VEL
LIN {X 0,Y 134.426,Z 457.021,A -85,B 0,C 180,E1 -26627.929,E2 -26627.929} C_VEL
LIN {X 0,Y 132.152,Z 452.059,A -85,B 0,C 180,E1 -26638.867,E2 -26638.867} C_VEL
LIN {X 0,Y 132.149,Z 452.347,A -85,B 0,C 180,E1 -26641.453,E2 -26641.453} C_VEL
LIN {X 0,Y 134.22,Z 456.875,A -85,B 0,C 180,E1 -26651.324,E2 -26651.324} C_VEL
LIN {X 0,Y 134.984,Z 457.732,A -85,B 0,C 180,E1 -26653.023,E2 -26653.023} C_VEL
LIN {X 0,Y 137.022,Z 461.105,A -85,B 0,C 180,E1 -26656.876,E2 -26656.876} C_VEL
LIN {X 0,Y 138.049,Z 462.596,A -85,B 0,C 180,E1 -26658.457,E2 -26658.457} C_VEL
LIN {X 0,Y 140.923,Z 467.041,A -85,B 0,C 180,E1 -26662.254,E2 -26662.254} C_VEL
LIN {X 0,Y 144.437,Z 472.808,A -85,B 0,C 180,E1 -26666.068,E2 -26666.068} C_VEL
LIN {X 0,Y 146.735,Z 477.639,A -85,B 0,C 180,E1 -26668.325,E2 -26668.325} C_VEL
LIN {X 0,Y 150.192,Z 486.484,A -85,B 0,C 180,E1 -26671.469,E2 -26671.469} C_VEL
LIN {X 0,Y 152.642,Z 493.727,A -85,B 0,C 180,E1 -26673.539,E2 -26673.539} C_VEL
LIN {X 0,Y 150.09,Z 521.668,A -85,B 0,C 180,E1 -26674.593,E2 -26674.593} C_VEL
LIN {X 0,Y 147.642,Z 535.326,A -85,B 0,C 180,E1 -26675.46,E2 -26675.46} C_VEL
LIN {X 0,Y 144.417,Z 547.361,A -85,B 0,C 180,E1 -26676.585,E2 -26676.585} C_VEL
LIN {X 0,Y 139.892,Z 560.007,A -85,B 0,C 180,E1 -26678.28,E2 -26678.28} C_VEL
LIN {X 0,Y 134.856,Z 571.259,A -85,B 0,C 180,E1 -26680.342,E2 -26680.342} C_VEL
LIN {X 0,Y 129.54,Z 581.396,A -85,B 0,C 180,E1 -26682.909,E2 -26682.909} C_VEL
LIN {X 0,Y 123.921,Z 590.533,A -85,B 0,C 180,E1 -26685.992,E2 -26685.992} C_VEL
LIN {X 0,Y 117.744,Z 599.442,A -85,B 0,C 180,E1 -26690.084,E2 -26690.084} C_VEL
LIN {X 0,Y 113.033,Z 605.871,A -85,B 0,C 180,E1 -26694.156,E2 -26694.156} C_VEL
LIN {X 0,Y 108.442,Z 611.457,A -85,B 0,C 180,E1 -26698.769,E2 -26698.769} C_VEL
LIN {X 0,Y 104.423,Z 616.164,A -85,B 0,C 180,E1 -26704.056,E2 -26704.056} C_VEL
LIN {X 0,Y 101.31,Z 619.762,A -85,B 0,C 180,E1 -26709.704,E2 -26709.704} C_VEL
LIN {X 0,Y 99.87,Z 621.62,A -85,B 0,C 180,E1 -26713.65,E2 -26713.65} C_VEL
LIN {X 0,Y 98.187,Z 624.012,A -85,B 0,C 180,E1 -26721.769,E2 -26721.769} C_VEL
LIN {X 0,Y 97.941,Z 624.622,A -85,B 0,C 180,E1 -26725.884,E2 -26725.884} C_VEL
LIN {X 0,Y 98.007,Z 624.835,A -85,B 0,C 180,E1 -26729.999,E2 -26729.999} C_VEL
LIN {X 0,Y 97.942,Z 624.604,A -85,B 0,C 180,E1 -26734.114,E2 -26734.114} C_VEL
LIN {X 0,Y 98.187,Z 623.984,A -85,B 0,C 180,E1 -26738.23,E2 -26738.23} C_VEL
LIN {X 0,Y 98.822,Z 622.975,A -85,B 0,C 180,E1 -26742.318,E2 -26742.318} C_VEL
LIN {X 0,Y 99.868,Z 621.564,A -85,B 0,C 180,E1 -26746.348,E2 -26746.348} C_VEL
LIN {X 0,Y 102.223,Z 618.61,A -85,B 0,C 180,E1 -26752.217,E2 -26752.217} C_VEL
LIN {X 0,Y 105.698,Z 614.624,A -85,B 0,C 180,E1 -26757.738,E2 -26757.738} C_VEL
LIN {X 0,Y 110.852,Z 608.498,A -85,B 0,C 180,E1 -26763.693,E2 -26763.693} C_VEL
LIN {X 0,Y 115.847,Z 601.804,A -85,B 0,C 180,E1 -26768.449,E2 -26768.449} C_VEL
LIN {X 0,Y 121.787,Z 593.513,A -85,B 0,C 180,E1 -26772.692,E2 -26772.692} C_VEL
LIN {X 0,Y 127.209,Z 585.005,A -85,B 0,C 180,E1 -26775.907,E2 -26775.907} C_VEL
LIN {X 0,Y 133.046,Z 574.498,A -85,B 0,C 180,E1 -26778.828,E2 -26778.828} C_VEL
LIN {X 0,Y 137.946,Z 564.098,A -85,B 0,C 180,E1 -26780.982,E2 -26780.982} C_VEL
LIN {X 0,Y 142.409,Z 552.683,A -85,B 0,C 180,E1 -26782.729,E2 -26782.729} C_VEL
LIN {X 0,Y 143.812,Z 548.399,A -85,B 0,C 180,E1 -26783.252,E2 -26783.252} C_VEL
LIN {X 0,Y 144.626,Z 544.787,A -85,B 0,C 180,E1 -26783.833,E2 -26783.833} C_VEL
LIN {X 0,Y 144.529,Z 539.128,A -85,B 0,C 180,E1 -26785.309,E2 -26785.309} C_VEL
LIN {X 0,Y 144.21,Z 533.352,A -85,B 0,C 180,E1 -26786.722,E2 -26786.722} C_VEL
LIN {X 0,Y 144.613,Z 529.549,A -85,B 0,C 180,E1 -26787.181,E2 -26787.181} C_VEL
LIN {X 0,Y 146.618,Z 515.974,A -85,B 0,C 180,E1 -26787.872,E2 -26787.872} C_VEL
LIN {X 0,Y 148.396,Z 495.866,A -85,B 0,C 180,E1 -26788.604,E2 -26788.604} C_VEL
LIN {X 0,Y 145.206,Z 486.543,A -85,B 0,C 180,E1 -26791.646,E2 -26791.646} C_VEL
LIN {X 0,Y 142.379,Z 479.514,A -85,B 0,C 180,E1 -26794.606,E2 -26794.606} C_VEL
LIN {X 0,Y 139.279,Z 474.005,A -85,B 0,C 180,E1 -26798.145,E2 -26798.145} C_VEL
LIN {X 0,Y 137.435,Z 470.975,A -85,B 0,C 180,E1 -26800.586,E2 -26800.586} C_VEL
LIN {X 0,Y 135.492,Z 467.753,A -85,B 0,C 180,E1 -26803.618,E2 -26803.618} C_VEL
LIN {X 0,Y 133.234,Z 463.961,A -85,B 0,C 180,E1 -26808.206,E2 -26808.206} C_VEL
LIN {X 0,Y 131.144,Z 460.373,A -85,B 0,C 180,E1 -26815.871,E2 -26815.871} C_VEL
LIN {X 0,Y 130.991,Z 459.07,A -85,B 0,C 180,E1 -26818.463,E2 -26818.463} C_VEL
LIN {X 0,Y 131.019,Z 459.225,A -85,B 0,C 180,E1 -26822.498,E2 -26822.498} C_VEL
LIN {X 0,Y 132.937,Z 463.689,A -85,B 0,C 180,E1 -26831.477,E2 -26831.477} C_VEL
LIN {X 0,Y 133.598,Z 464.509,A -85,B 0,C 180,E1 -26833.016,E2 -26833.016} C_VEL
LIN {X 0,Y 136.38,Z 469.162,A -85,B 0,C 180,E1 -26838.205,E2 -26838.205} C_VEL
LIN {X 0,Y 138.954,Z 473.461,A -85,B 0,C 180,E1 -26841.823,E2 -26841.823} C_VEL
LIN {X 0,Y 142.126,Z 478.951,A -85,B 0,C 180,E1 -26845.491,E2 -26845.491} C_VEL
LIN {X 0,Y 146.234,Z 487.057,A -85,B 0,C 180,E1 -26849.513,E2 -26849.513} C_VEL
LIN {X 0,Y 148.644,Z 492.304,A -85,B 0,C 180,E1 -26851.606,E2 -26851.606} C_VEL
LIN {X 0,Y 147.798,Z 503.06,A -85,B 0,C 180,E1 -26852.049,E2 -26852.049} C_VEL
LIN {X 0,Y 146.069,Z 519.277,A -85,B 0,C 180,E1 -26852.689,E2 -26852.689} C_VEL
LIN {X 0,Y 143.822,Z 531.269,A -85,B 0,C 180,E1 -26853.474,E2 -26853.474} C_VEL
LIN {X 0,Y 140.438,Z 543.691,A -85,B 0,C 180,E1 -26854.656,E2 -26854.656} C_VEL
LIN {X 0,Y 136.266,Z 555.468,A -85,B 0,C 180,E1 -26856.306,E2 -26856.306} C_VEL
LIN {X 0,Y 131.174,Z 566.795,A -85,B 0,C 180,E1 -26858.411,E2 -26858.411} C_VEL
LIN {X 0,Y 125.678,Z 577,A -85,B 0,C 180,E1 -26860.981,E2 -26860.981} C_VEL
LIN {X 0,Y 119.917,Z 586.16,A -85,B 0,C 180,E1 -26864.116,E2 -26864.116} C_VEL
LIN {X 0,Y 113.611,Z 595.061,A -85,B 0,C 180,E1 -26868.319,E2 -26868.319} C_VEL
LIN {X 0,Y 107.858,Z 602.225,A -85,B 0,C 180,E1 -26872.935,E2 -26872.935} C_VEL
LIN {X 0,Y 103.497,Z 607.056,A -85,B 0,C 180,E1 -26877.096,E2 -26877.096} C_VEL
LIN {X 0,Y 99.078,Z 611.747,A -85,B 0,C 180,E1 -26882.544,E2 -26882.544} C_VEL
LIN {X 0,Y 95.61,Z 615.333,A -85,B 0,C 180,E1 -26888.437,E2 -26888.437} C_VEL
LIN {X 0,Y 93.847,Z 617.183,A -85,B 0,C 180,E1 -26892.57,E2 -26892.57} C_VEL
LIN {X 0,Y 91.562,Z 619.558,A -85,B 0,C 180,E1 -26901.17,E2 -26901.17} C_VEL
LIN {X 0,Y 91.106,Z 620.161,A -85,B 0,C 180,E1 -26905.577,E2 -26905.577} C_VEL
LIN {X 0,Y 91.003,Z 620.385,A -85,B 0,C 180,E1 -26910.001,E2 -26910.001} C_VEL
LIN {X 0,Y 91.107,Z 620.188,A -85,B 0,C 180,E1 -26914.425,E2 -26914.425} C_VEL
LIN {X 0,Y 92.449,Z 618.633,A -85,B 0,C 180,E1 -26923.184,E2 -26923.184} C_VEL
LIN {X 0,Y 93.845,Z 617.272,A -85,B 0,C 180,E1 -26927.432,E2 -26927.432} C_VEL
LIN {X 0,Y 96.632,Z 614.398,A -85,B 0,C 180,E1 -26933.58,E2 -26933.58} C_VEL
LIN {X 0,Y 100.335,Z 610.5,A -85,B 0,C 180,E1 -26939.363,E2 -26939.363} C_VEL
LIN {X 0,Y 105.123,Z 605.464,A -85,B 0,C 180,E1 -26944.631,E2 -26944.631} C_VEL
LIN {X 0,Y 110.541,Z 599.124,A -85,B 0,C 180,E1 -26949.479,E2 -26949.479} C_VEL
LIN {X 0,Y 116.377,Z 591.491,A -85,B 0,C 180,E1 -26953.748,E2 -26953.748} C_VEL
LIN {X 0,Y 122.082,Z 583.109,A -85,B 0,C 180,E1 -26957.223,E2 -26957.223} C_VEL
LIN {X 0,Y 128.05,Z 573.236,A -85,B 0,C 180,E1 -26960.21,E2 -26960.21} C_VEL
LIN {X 0,Y 133.617,Z 562.113,A -85,B 0,C 180,E1 -26962.708,E2 -26962.708} C_VEL
LIN {X 0,Y 138.092,Z 551.208,A -85,B 0,C 180,E1 -26964.519,E2 -26964.519} C_VEL
LIN {X 0,Y 142.051,Z 539.144,A -85,B 0,C 180,E1 -26965.968,E2 -26965.968} C_VEL
LIN {X 0,Y 145.065,Z 526.515,A -85,B 0,C 180,E1 -26967.037,E2 -26967.037} C_VEL
LIN {X 0,Y 147.036,Z 513.671,A -85,B 0,C 180,E1 -26967.715,E2 -26967.715} C_VEL
LIN {X 0,Y 148.939,Z 492.699,A -85,B 0,C 180,E1 -26968.469,E2 -26968.469} C_VEL
LIN {X 0,Y 144.911,Z 484.032,A -85,B 0,C 180,E1 -26972.075,E2 -26972.075} C_VEL
LIN {X 0,Y 141.436,Z 477.565,A -85,B 0,C 180,E1 -26975.652,E2 -26975.652} C_VEL
LIN {X 0,Y 138.273,Z 472.066,A -85,B 0,C 180,E1 -26979.547,E2 -26979.547} C_VEL
LIN {X 0,Y 135.711,Z 467.92,A -85,B 0,C 180,E1 -26983.451,E2 -26983.451} C_VEL
LIN {X 0,Y 133.577,Z 464.092,A -85,B 0,C 180,E1 -26987.851,E2 -26987.851} C_VEL
LIN {X 0,Y 131.273,Z 459.785,A -85,B 0,C 180,E1 -26997.753,E2 -26997.753} C_VEL
LIN {X 0,Y 131.277,Z 459.082,A -85,B 0,C 180,E1 -26999.287,E2 -26999.287} C_VEL
LIN {X 0,Y 131.262,Z 459.428,A -85,B 0,C 180,E1 -27001.17,E2 -27001.17} C_VEL
LIN {X 0,Y 133.361,Z 464.018,A -85,B 0,C 180,E1 -27011.398,E2 -27011.398} C_VEL
LIN {X 0,Y 133.895,Z 464.974,A -85,B 0,C 180,E1 -27012.697,E2 -27012.697} C_VEL
LIN {X 0,Y 136.358,Z 468.964,A -85,B 0,C 180,E1 -27017.342,E2 -27017.342} C_VEL
LIN {X 0,Y 139.183,Z 473.665,A -85,B 0,C 180,E1 -27021.377,E2 -27021.377} C_VEL
LIN {X 0,Y 142.23,Z 478.978,A -85,B 0,C 180,E1 -27024.93,E2 -27024.93} C_VEL
LIN {X 0,Y 144.716,Z 484.803,A -85,B 0,C 180,E1 -27027.573,E2 -27027.573} C_VEL
LIN {X 0,Y 148.314,Z 495.113,A -85,B 0,C 180,E1 -27031.069,E2 -27031.069} C_VEL
LIN {X 0,Y 148.613,Z 496.073,A -85,B 0,C 180,E1 -27031.345,E2 -27031.345} C_VEL
LIN {X 0,Y 146.202,Z 521.396,A -85,B 0,C 180,E1 -27032.3,E2 -27032.3} C_VEL
LIN {X 0,Y 143.694,Z 534.87,A -85,B 0,C 180,E1 -27033.123,E2 -27033.123} C_VEL
LIN {X 0,Y 140.306,Z 547.201,A -85,B 0,C 180,E1 -27034.258,E2 -27034.258} C_VEL
LIN {X 0,Y 135.609,Z 559.845,A -85,B 0,C 180,E1 -27035.925,E2 -27035.925} C_VEL
LIN {X 0,Y 130.366,Z 571.096,A -85,B 0,C 180,E1 -27037.96,E2 -27037.96} C_VEL
LIN {X 0,Y 124.803,Z 581.232,A -85,B 0,C 180,E1 -27040.515,E2 -27040.515} C_VEL
LIN {X 0,Y 118.891,Z 590.367,A -85,B 0,C 180,E1 -27043.602,E2 -27043.602} C_VEL
LIN {X 0,Y 112.382,Z 599.276,A -85,B 0,C 180,E1 -27047.756,E2 -27047.756} C_VEL
LIN {X 0,Y 106.887,Z 606.253,A -85,B 0,C 180,E1 -27052.324,E2 -27052.324} C_VEL
LIN {X 0,Y 102.427,Z 611.291,A -85,B 0,C 180,E1 -27056.706,E2 -27056.706} C_VEL
LIN {X 0,Y 98.063,Z 615.997,A -85,B 0,C 180,E1 -27062.234,E2 -27062.234} C_VEL
LIN {X 0,Y 94.645,Z 619.594,A -85,B 0,C 180,E1 -27068.204,E2 -27068.204} C_VEL
LIN {X 0,Y 93.042,Z 621.452,A -85,B 0,C 180,E1 -27072.413,E2 -27072.413} C_VEL
LIN {X 0,Y 91.874,Z 622.846,A -85,B 0,C 180,E1 -27076.732,E2 -27076.732} C_VEL
LIN {X 0,Y 90.871,Z 624.455,A -85,B 0,C 180,E1 -27085.563,E2 -27085.563} C_VEL
LIN {X 0,Y 90.913,Z 624.668,A -85,B 0,C 180,E1 -27089.999,E2 -27089.999} C_VEL
LIN {X 0,Y 90.871,Z 624.437,A -85,B 0,C 180,E1 -27094.435,E2 -27094.435} C_VEL
LIN {X 0,Y 91.874,Z 622.807,A -85,B 0,C 180,E1 -27103.266,E2 -27103.266} C_VEL
LIN {X 0,Y 93.041,Z 621.395,A -85,B 0,C 180,E1 -27107.586,E2 -27107.586} C_VEL
LIN {X 0,Y 95.676,Z 618.442,A -85,B 0,C 180,E1 -27113.828,E2 -27113.828} C_VEL
LIN {X 0,Y 99.457,Z 614.455,A -85,B 0,C 180,E1 -27119.646,E2 -27119.646} C_VEL
LIN {X 0,Y 104.99,Z 608.328,A -85,B 0,C 180,E1 -27125.853,E2 -27125.853} C_VEL
LIN {X 0,Y 110.349,Z 601.634,A -85,B 0,C 180,E1 -27130.753,E2 -27130.753} C_VEL
LIN {X 0,Y 116.647,Z 593.343,A -85,B 0,C 180,E1 -27135.067,E2 -27135.067} C_VEL
LIN {X 0,Y 122.371,Z 584.835,A -85,B 0,C 180,E1 -27138.297,E2 -27138.297} C_VEL
LIN {X 0,Y 128.484,Z 574.327,A -85,B 0,C 180,E1 -27141.211,E2 -27141.211} C_VEL
LIN {X 0,Y 134.246,Z 562.494,A -85,B 0,C 180,E1 -27143.601,E2 -27143.601} C_VEL
LIN {X 0,Y 138.882,Z 550.557,A -85,B 0,C 180,E1 -27145.317,E2 -27145.317} C_VEL
LIN {X 0,Y 142.715,Z 538.13,A -85,B 0,C 180,E1 -27146.52,E2 -27146.52} C_VEL
LIN {X 0,Y 144.613,Z 529.549,A -85,B 0,C 180,E1 -27147.181,E2 -27147.181} C_VEL
LIN {X 0,Y 144.998,Z 525.732,A -85,B 0,C 180,E1 -27147.612,E2 -27147.612} C_VEL
LIN {X 0,Y 144.359,Z 519.811,A -85,B 0,C 180,E1 -27148.88,E2 -27148.88} C_VEL
LIN {X 0,Y 143.52,Z 513.85,A -85,B 0,C 180,E1 -27150.119,E2 -27150.119} C_VEL
LIN {X 0,Y 143.547,Z 509.965,A -85,B 0,C 180,E1 -27150.482,E2 -27150.482} C_VEL
LIN {X 0,Y 144.565,Z 498.42,A -85,B 0,C 180,E1 -27150.912,E2 -27150.912} C_VEL
LIN {X 0,Y 141.676,Z 489.692,A -85,B 0,C 180,E1 -27154.036,E2 -27154.036} C_VEL
LIN {X 0,Y 139.613,Z 484.42,A -85,B 0,C 180,E1 -27156.469,E2 -27156.469} C_VEL
LIN {X 0,Y 136.422,Z 478.451,A -85,B 0,C 180,E1 -27160.632,E2 -27160.632} C_VEL
LIN {X 0,Y 133.987,Z 474.323,A -85,B 0,C 180,E1 -27164.601,E2 -27164.601} C_VEL
LIN {X 0,Y 132.056,Z 470.803,A -85,B 0,C 180,E1 -27168.877,E2 -27168.877} C_VEL
LIN {X 0,Y 130.18,Z 467.147,A -85,B 0,C 180,E1 -27176.712,E2 -27176.712} C_VEL
LIN {X 0,Y 130.117,Z 466.19,A -85,B 0,C 180,E1 -27178.453,E2 -27178.453} C_VEL
LIN {X 0,Y 130.122,Z 466.156,A -85,B 0,C 180,E1 -27181.935,E2 -27181.935} C_VEL
LIN {X 0,Y 131.881,Z 470.647,A -85,B 0,C 180,E1 -27191.069,E2 -27191.069} C_VEL
LIN {X 0,Y 132.446,Z 471.575,A -85,B 0,C 180,E1 -27192.508,E2 -27192.508} C_VEL
LIN {X 0,Y 134.761,Z 475.661,A -85,B 0,C 180,E1 -27197.157,E2 -27197.157} C_VEL
LIN {X 0,Y 137.17,Z 479.918,A -85,B 0,C 180,E1 -27200.821,E2 -27200.821} C_VEL
LIN {X 0,Y 140.008,Z 485.177,A -85,B 0,C 180,E1 -27204.366,E2 -27204.366} C_VEL
LIN {X 0,Y 143.671,Z 492.943,A -85,B 0,C 180,E1 -27208.257,E2 -27208.257} C_VEL
LIN {X 0,Y 144.82,Z 495.621,A -85,B 0,C 180,E1 -27209.366,E2 -27209.366} C_VEL
LIN {X 0,Y 142.513,Z 518.349,A -85,B 0,C 180,E1 -27210.218,E2 -27210.218} C_VEL
LIN {X 0,Y 140.002,Z 531.598,A -85,B 0,C 180,E1 -27211.065,E2 -27211.065} C_VEL
LIN {X 0,Y 136.537,Z 543.865,A -85,B 0,C 180,E1 -27212.211,E2 -27212.211} C_VEL
LIN {X 0,Y 132.193,Z 555.64,A -85,B 0,C 180,E1 -27213.83,E2 -27213.83} C_VEL
LIN {X 0,Y 126.899,Z 566.965,A -85,B 0,C 180,E1 -27215.907,E2 -27215.907} C_VEL
LIN {X 0,Y 121.152,Z 577.17,A -85,B 0,C 180,E1 -27218.453,E2 -27218.453} C_VEL
LIN {X 0,Y 115.078,Z 586.33,A -85,B 0,C 180,E1 -27221.572,E2 -27221.572} C_VEL
LIN {X 0,Y 108.415,Z 595.23,A -85,B 0,C 180,E1 -27225.824,E2 -27225.824} C_VEL
LIN {X 0,Y 102.292,Z 602.393,A -85,B 0,C 180,E1 -27230.542,E2 -27230.542} C_VEL
LIN {X 0,Y 97.611,Z 607.224,A -85,B 0,C 180,E1 -27234.831,E2 -27234.831} C_VEL
LIN {X 0,Y 92.826,Z 611.916,A -85,B 0,C 180,E1 -27240.52,E2 -27240.52} C_VEL
LIN {X 0,Y 89.039,Z 615.501,A -85,B 0,C 180,E1 -27246.756,E2 -27246.756} C_VEL
LIN {X 0,Y 87.082,Z 617.351,A -85,B 0,C 180,E1 -27251.167,E2 -27251.167} C_VEL
LIN {X 0,Y 85.563,Z 618.739,A -85,B 0,C 180,E1 -27255.735,E2 -27255.735} C_VEL
LIN {X 0,Y 84.051,Z 620.328,A -85,B 0,C 180,E1 -27265.204,E2 -27265.204} C_VEL
LIN {X 0,Y 83.923,Z 620.551,A -85,B 0,C 180,E1 -27270.001,E2 -27270.001} C_VEL
LIN {X 0,Y 84.051,Z 620.355,A -85,B 0,C 180,E1 -27274.797,E2 -27274.797} C_VEL
LIN {X 0,Y 85.564,Z 618.8,A -85,B 0,C 180,E1 -27284.266,E2 -27284.266} C_VEL
LIN {X 0,Y 87.079,Z 617.439,A -85,B 0,C 180,E1 -27288.835,E2 -27288.835} C_VEL
LIN {X 0,Y 90.151,Z 614.565,A -85,B 0,C 180,E1 -27295.39,E2 -27295.39} C_VEL
LIN {X 0,Y 94.198,Z 610.667,A -85,B 0,C 180,E1 -27301.485,E2 -27301.485} C_VEL
LIN {X 0,Y 99.358,Z 605.63,A -85,B 0,C 180,E1 -27306.96,E2 -27306.96} C_VEL
LIN {X 0,Y 105.149,Z 599.289,A -85,B 0,C 180,E1 -27311.944,E2 -27311.944} C_VEL
LIN {X 0,Y 111.352,Z 591.656,A -85,B 0,C 180,E1 -27316.277,E2 -27316.277} C_VEL
LIN {X 0,Y 117.379,Z 583.273,A -85,B 0,C 180,E1 -27319.766,E2 -27319.766} C_VEL
LIN {X 0,Y 123.634,Z 573.4,A -85,B 0,C 180,E1 -27322.735,E2 -27322.735} C_VEL
LIN {X 0,Y 129.439,Z 562.275,A -85,B 0,C 180,E1 -27325.209,E2 -27325.209} C_VEL
LIN {X 0,Y 134.105,Z 551.369,A -85,B 0,C 180,E1 -27326.984,E2 -27326.984} C_VEL
LIN {X 0,Y 138.215,Z 539.303,A -85,B 0,C 180,E1 -27328.4,E2 -27328.4} C_VEL
LIN {X 0,Y 141.384,Z 526.415,A -85,B 0,C 180,E1 -27329.463,E2 -27329.463} C_VEL
LIN {X 0,Y 143.513,Z 512.576,A -85,B 0,C 180,E1 -27330.16,E2 -27330.16} C_VEL
LIN {X 0,Y 144.996,Z 496.448,A -85,B 0,C 180,E1 -27330.748,E2 -27330.748} C_VEL
LIN {X 0,Y 144.844,Z 495.28,A -85,B 0,C 180,E1 -27330.973,E2 -27330.973} C_VEL
LIN {X 0,Y 141.144,Z 487.166,A -85,B 0,C 180,E1 -27334.763,E2 -27334.763} C_VEL
LIN {X 0,Y 138.078,Z 481.264,A -85,B 0,C 180,E1 -27338.444,E2 -27338.444} C_VEL
LIN {X 0,Y 135.967,Z 477.644,A -85,B 0,C 180,E1 -27341.425,E2 -27341.425} C_VEL
LIN {X 0,Y 134.151,Z 474.397,A -85,B 0,C 180,E1 -27344.546,E2 -27344.546} C_VEL
LIN {X 0,Y 132.236,Z 470.88,A -85,B 0,C 180,E1 -27348.892,E2 -27348.892} C_VEL
LIN {X 0,Y 130.406,Z 466.125,A -85,B 0,C 180,E1 -27360,E2 -27360} C_VEL
LIN {X 0,Y 132.48,Z 471.334,A -85,B 0,C 180,E1 -27371.475,E2 -27371.475} C_VEL
LIN {X 0,Y 134.84,Z 475.586,A -85,B 0,C 180,E1 -27376.422,E2 -27376.422} C_VEL
LIN {X 0,Y 137.291,Z 479.89,A -85,B 0,C 180,E1 -27380.214,E2 -27380.214} C_VEL
LIN {X 0,Y 140.09,Z 485.125,A -85,B 0,C 180,E1 -27383.762,E2 -27383.762} C_VEL
LIN {X 0,Y 142.477,Z 491.51,A -85,B 0,C 180,E1 -27386.553,E2 -27386.553} C_VEL
LIN {X 0,Y 144.791,Z 498.634,A -85,B 0,C 180,E1 -27389.038,E2 -27389.038} C_VEL
LIN {X 0,Y 142.513,Z 521.439,A -85,B 0,C 180,E1 -27389.903,E2 -27389.903} C_VEL
LIN {X 0,Y 139.857,Z 535.067,A -85,B 0,C 180,E1 -27390.712,E2 -27390.712} C_VEL
LIN {X 0,Y 136.436,Z 547.04,A -85,B 0,C 180,E1 -27391.793,E2 -27391.793} C_VEL
LIN {X 0,Y 131.567,Z 559.683,A -85,B 0,C 180,E1 -27393.419,E2 -27393.419} C_VEL
LIN {X 0,Y 126.126,Z 570.933,A -85,B 0,C 180,E1 -27395.418,E2 -27395.418} C_VEL
LIN {X 0,Y 120.311,Z 581.068,A -85,B 0,C 180,E1 -27397.943,E2 -27397.943} C_VEL
LIN {X 0,Y 114.093,Z 590.202,A -85,B 0,C 180,E1 -27401.01,E2 -27401.01} C_VEL
LIN {X 0,Y 107.217,Z 599.111,A -85,B 0,C 180,E1 -27405.197,E2 -27405.197} C_VEL
LIN {X 0,Y 101.581,Z 605.724,A -85,B 0,C 180,E1 -27409.557,E2 -27409.557} C_VEL
LIN {X 0,Y 96.566,Z 611.125,A -85,B 0,C 180,E1 -27414.391,E2 -27414.391} C_VEL
LIN {X 0,Y 91.823,Z 615.831,A -85,B 0,C 180,E1 -27420.164,E2 -27420.164} C_VEL
LIN {X 0,Y 88.059,Z 619.427,A -85,B 0,C 180,E1 -27426.48,E2 -27426.48} C_VEL
LIN {X 0,Y 86.273,Z 621.285,A -85,B 0,C 180,E1 -27430.982,E2 -27430.982} C_VEL
LIN {X 0,Y 84.965,Z 622.679,A -85,B 0,C 180,E1 -27435.631,E2 -27435.631} C_VEL
LIN {X 0,Y 83.787,Z 624.288,A -85,B 0,C 180,E1 -27445.187,E2 -27445.187} C_VEL
LIN {X 0,Y 83.812,Z 624.501,A -85,B 0,C 180,E1 -27449.999,E2 -27449.999} C_VEL
LIN {X 0,Y 83.787,Z 624.27,A -85,B 0,C 180,E1 -27454.811,E2 -27454.811} C_VEL
LIN {X 0,Y 84.964,Z 622.639,A -85,B 0,C 180,E1 -27464.367,E2 -27464.367} C_VEL
LIN {X 0,Y 86.272,Z 621.226,A -85,B 0,C 180,E1 -27469.017,E2 -27469.017} C_VEL
LIN {X 0,Y 89.192,Z 618.273,A -85,B 0,C 180,E1 -27475.682,E2 -27475.682} C_VEL
LIN {X 0,Y 93.321,Z 614.286,A -85,B 0,C 180,E1 -27481.814,E2 -27481.814} C_VEL
LIN {X 0,Y 99.274,Z 608.158,A -85,B 0,C 180,E1 -27488.275,E2 -27488.275} C_VEL
LIN {X 0,Y 105.045,Z 601.464,A -85,B 0,C 180,E1 -27493.296,E2 -27493.296} C_VEL
LIN {X 0,Y 111.738,Z 593.173,A -85,B 0,C 180,E1 -27497.649,E2 -27497.649} C_VEL
LIN {X 0,Y 117.77,Z 584.665,A -85,B 0,C 180,E1 -27500.875,E2 -27500.875} C_VEL
LIN {X 0,Y 124.15,Z 574.156,A -85,B 0,C 180,E1 -27503.772,E2 -27503.772} C_VEL
LIN {X 0,Y 130.157,Z 562.322,A -85,B 0,C 180,E1 -27506.118,E2 -27506.118} C_VEL
LIN {X 0,Y 134.972,Z 550.383,A -85,B 0,C 180,E1 -27507.794,E2 -27507.794} C_VEL
LIN {X 0,Y 138.929,Z 537.955,A -85,B 0,C 180,E1 -27508.961,E2 -27508.961} C_VEL
LIN {X 0,Y 141.651,Z 525.515,A -85,B 0,C 180,E1 -27509.824,E2 -27509.824} C_VEL
LIN {X 0,Y 143.412,Z 511.307,A -85,B 0,C 180,E1 -27510.444,E2 -27510.444} C_VEL
LIN {X 0,Y 143.547,Z 509.965,A -85,B 0,C 180,E1 -27510.482,E2 -27510.482} C_VEL
LIN {X 0,Y 143.518,Z 506.876,A -85,B 0,C 180,E1 -27510.81,E2 -27510.81} C_VEL
LIN {X 0,Y 142.674,Z 503.124,A -85,B 0,C 180,E1 -27511.805,E2 -27511.805} C_VEL
LIN {X 0,Y 140.288,Z 497.844,A -85,B 0,C 180,E1 -27514.263,E2 -27514.263} C_VEL
LIN {X 0,Y 138.828,Z 494.209,A -85,B 0,C 180,E1 -27515.977,E2 -27515.977} C_VEL
LIN {X 0,Y 137.249,Z 489.984,A -85,B 0,C 180,E1 -27518.055,E2 -27518.055} C_VEL
LIN {X 0,Y 134.575,Z 484.659,A -85,B 0,C 180,E1 -27521.916,E2 -27521.916} C_VEL
LIN {X 0,Y 132.49,Z 480.837,A -85,B 0,C 180,E1 -27525.669,E2 -27525.669} C_VEL
LIN {X 0,Y 130.892,Z 477.681,A -85,B 0,C 180,E1 -27529.56,E2 -27529.56} C_VEL
LIN {X 0,Y 129.225,Z 473.578,A -85,B 0,C 180,E1 -27538.247,E2 -27538.247} C_VEL
LIN {X 0,Y 129.216,Z 473.047,A -85,B 0,C 180,E1 -27540,E2 -27540} C_VEL
LIN {X 0,Y 129.243,Z 473.5,A -85,B 0,C 180,E1 -27542.24,E2 -27542.24} C_VEL
LIN {X 0,Y 130.761,Z 477.517,A -85,B 0,C 180,E1 -27550.456,E2 -27550.456} C_VEL
LIN {X 0,Y 131.376,Z 478.767,A -85,B 0,C 180,E1 -27552.171,E2 -27552.171} C_VEL
LIN {X 0,Y 133.194,Z 482.121,A -85,B 0,C 180,E1 -27556.082,E2 -27556.082} C_VEL
LIN {X 0,Y 135.44,Z 486.411,A -85,B 0,C 180,E1 -27559.811,E2 -27559.811} C_VEL
LIN {X 0,Y 138.103,Z 491.786,A -85,B 0,C 180,E1 -27563.409,E2 -27563.409} C_VEL
LIN {X 0,Y 141.205,Z 498.875,A -85,B 0,C 180,E1 -27566.982,E2 -27566.982} C_VEL
LIN {X 0,Y 139.09,Z 518.453,A -85,B 0,C 180,E1 -27567.688,E2 -27567.688} C_VEL
LIN {X 0,Y 136.456,Z 531.874,A -85,B 0,C 180,E1 -27568.523,E2 -27568.523} C_VEL
LIN {X 0,Y 132.888,Z 544.038,A -85,B 0,C 180,E1 -27569.62,E2 -27569.62} C_VEL
LIN {X 0,Y 128.382,Z 555.812,A -85,B 0,C 180,E1 -27571.202,E2 -27571.202} C_VEL
LIN {X 0,Y 122.872,Z 567.137,A -85,B 0,C 180,E1 -27573.226,E2 -27573.226} C_VEL
LIN {X 0,Y 116.882,Z 577.34,A -85,B 0,C 180,E1 -27575.734,E2 -27575.734} C_VEL
LIN {X 0,Y 110.498,Z 586.5,A -85,B 0,C 180,E1 -27578.819,E2 -27578.819} C_VEL
LIN {X 0,Y 103.824,Z 594.933,A -85,B 0,C 180,E1 -27582.817,E2 -27582.817} C_VEL
LIN {X 0,Y 96.924,Z 602.562,A -85,B 0,C 180,E1 -27587.878,E2 -27587.878} C_VEL
LIN {X 0,Y 91.886,Z 607.393,A -85,B 0,C 180,E1 -27592.275,E2 -27592.275} C_VEL
LIN {X 0,Y 86.69,Z 612.085,A -85,B 0,C 180,E1 -27598.201,E2 -27598.201} C_VEL
LIN {X 0,Y 82.542,Z 615.67,A -85,B 0,C 180,E1 -27604.804,E2 -27604.804} C_VEL
LIN {X 0,Y 80.387,Z 617.519,A -85,B 0,C 180,E1 -27609.532,E2 -27609.532} C_VEL
LIN {X 0,Y 78.695,Z 618.907,A -85,B 0,C 180,E1 -27614.46,E2 -27614.46} C_VEL
LIN {X 0,Y 76.988,Z 620.495,A -85,B 0,C 180,E1 -27624.763,E2 -27624.763} C_VEL
LIN {X 0,Y 76.843,Z 620.718,A -85,B 0,C 180,E1 -27630.001,E2 -27630.001} C_VEL
LIN {X 0,Y 76.989,Z 620.522,A -85,B 0,C 180,E1 -27635.239,E2 -27635.239} C_VEL
LIN {X 0,Y 78.696,Z 618.967,A -85,B 0,C 180,E1 -27645.542,E2 -27645.542} C_VEL
LIN {X 0,Y 80.384,Z 617.605,A -85,B 0,C 180,E1 -27650.471,E2 -27650.471} C_VEL
LIN {X 0,Y 83.779,Z 614.732,A -85,B 0,C 180,E1 -27657.477,E2 -27657.477} C_VEL
LIN {X 0,Y 88.213,Z 610.833,A -85,B 0,C 180,E1 -27663.898,E2 -27663.898} C_VEL
LIN {X 0,Y 93.781,Z 605.796,A -85,B 0,C 180,E1 -27669.57,E2 -27669.57} C_VEL
LIN {X 0,Y 99.978,Z 599.455,A -85,B 0,C 180,E1 -27674.666,E2 -27674.666} C_VEL
LIN {X 0,Y 106.806,Z 591.524,A -85,B 0,C 180,E1 -27679.177,E2 -27679.177} C_VEL
LIN {X 0,Y 112.929,Z 583.437,A -85,B 0,C 180,E1 -27682.513,E2 -27682.513} C_VEL
LIN {X 0,Y 119.47,Z 573.563,A -85,B 0,C 180,E1 -27685.445,E2 -27685.445} C_VEL
LIN {X 0,Y 125.534,Z 562.437,A -85,B 0,C 180,E1 -27687.864,E2 -27687.864} C_VEL
LIN {X 0,Y 130.382,Z 551.53,A -85,B 0,C 180,E1 -27689.595,E2 -27689.595} C_VEL
LIN {X 0,Y 134.637,Z 539.463,A -85,B 0,C 180,E1 -27690.97,E2 -27690.97} C_VEL
LIN {X 0,Y 137.867,Z 526.815,A -85,B 0,C 180,E1 -27691.988,E2 -27691.988} C_VEL
LIN {X 0,Y 140.052,Z 513.319,A -85,B 0,C 180,E1 -27692.652,E2 -27692.652} C_VEL
LIN {X 0,Y 141.447,Z 499.062,A -85,B 0,C 180,E1 -27693.154,E2 -27693.154} C_VEL
LIN {X 0,Y 138.36,Z 491.983,A -85,B 0,C 180,E1 -27696.72,E2 -27696.72} C_VEL
LIN {X 0,Y 135.635,Z 486.517,A -85,B 0,C 180,E1 -27700.416,E2 -27700.416} C_VEL
LIN {X 0,Y 134.086,Z 483.62,A -85,B 0,C 180,E1 -27702.902,E2 -27702.902} C_VEL
LIN {X 0,Y 132.756,Z 481.051,A -85,B 0,C 180,E1 -27705.436,E2 -27705.436} C_VEL
LIN {X 0,Y 131.088,Z 477.715,A -85,B 0,C 180,E1 -27709.575,E2 -27709.575} C_VEL
LIN {X 0,Y 129.528,Z 473.274,A -85,B 0,C 180,E1 -27720,E2 -27720} C_VEL
LIN {X 0,Y 131.306,Z 478.229,A -85,B 0,C 180,E1 -27730.797,E2 -27730.797} C_VEL
LIN {X 0,Y 133.46,Z 482.393,A -85,B 0,C 180,E1 -27735.672,E2 -27735.672} C_VEL
LIN {X 0,Y 135.751,Z 486.727,A -85,B 0,C 180,E1 -27739.468,E2 -27739.468} C_VEL
LIN {X 0,Y 138.197,Z 491.83,A -85,B 0,C 180,E1 -27742.816,E2 -27742.816} C_VEL
LIN {X 0,Y 140.458,Z 498.847,A -85,B 0,C 180,E1 -27745.721,E2 -27745.721} C_VEL
LIN {X 0,Y 141.194,Z 501.39,A -85,B 0,C 180,E1 -27746.614,E2 -27746.614} C_VEL
LIN {X 0,Y 139.009,Z 521.906,A -85,B 0,C 180,E1 -27747.394,E2 -27747.394} C_VEL
LIN {X 0,Y 136.419,Z 534.673,A -85,B 0,C 180,E1 -27748.126,E2 -27748.126} C_VEL
LIN {X 0,Y 132.837,Z 546.88,A -85,B 0,C 180,E1 -27749.193,E2 -27749.193} C_VEL
LIN {X 0,Y 127.8,Z 559.521,A -85,B 0,C 180,E1 -27750.765,E2 -27750.765} C_VEL
LIN {X 0,Y 122.137,Z 570.769,A -85,B 0,C 180,E1 -27752.694,E2 -27752.694} C_VEL
LIN {X 0,Y 116.076,Z 580.903,A -85,B 0,C 180,E1 -27755.176,E2 -27755.176} C_VEL
LIN {X 0,Y 109.561,Z 590.037,A -85,B 0,C 180,E1 -27758.204,E2 -27758.204} C_VEL
LIN {X 0,Y 102.279,Z 598.945,A -85,B 0,C 180,E1 -27762.38,E2 -27762.38} C_VEL
LIN {X 0,Y 95.815,Z 606.045,A -85,B 0,C 180,E1 -27767.18,E2 -27767.18} C_VEL
LIN {X 0,Y 90.884,Z 610.959,A -85,B 0,C 180,E1 -27771.782,E2 -27771.782} C_VEL
LIN {X 0,Y 85.721,Z 615.664,A -85,B 0,C 180,E1 -27777.796,E2 -27777.796} C_VEL
LIN {X 0,Y 81.566,Z 619.26,A -85,B 0,C 180,E1 -27784.479,E2 -27784.479} C_VEL
LIN {X 0,Y 79.574,Z 621.118,A -85,B 0,C 180,E1 -27789.311,E2 -27789.311} C_VEL
LIN {X 0,Y 77.123,Z 623.51,A -85,B 0,C 180,E1 -27799.498,E2 -27799.498} C_VEL
LIN {X 0,Y 76.708,Z 624.121,A -85,B 0,C 180,E1 -27804.742,E2 -27804.742} C_VEL
LIN {X 0,Y 76.733,Z 624.334,A -85,B 0,C 180,E1 -27809.999,E2 -27809.999} C_VEL
LIN {X 0,Y 76.708,Z 624.102,A -85,B 0,C 180,E1 -27815.256,E2 -27815.256} C_VEL
LIN {X 0,Y 78.07,Z 622.471,A -85,B 0,C 180,E1 -27825.667,E2 -27825.667} C_VEL
LIN {X 0,Y 79.572,Z 621.058,A -85,B 0,C 180,E1 -27830.688,E2 -27830.688} C_VEL
LIN {X 0,Y 82.826,Z 618.104,A -85,B 0,C 180,E1 -27837.819,E2 -27837.819} C_VEL
LIN {X 0,Y 87.326,Z 614.117,A -85,B 0,C 180,E1 -27844.288,E2 -27844.288} C_VEL
LIN {X 0,Y 93.758,Z 607.988,A -85,B 0,C 180,E1 -27850.986,E2 -27850.986} C_VEL
LIN {X 0,Y 99.988,Z 601.295,A -85,B 0,C 180,E1 -27856.091,E2 -27856.091} C_VEL
LIN {X 0,Y 107.082,Z 593.003,A -85,B 0,C 180,E1 -27860.459,E2 -27860.459} C_VEL
LIN {X 0,Y 113.419,Z 584.495,A -85,B 0,C 180,E1 -27863.662,E2 -27863.662} C_VEL
LIN {X 0,Y 120.095,Z 573.985,A -85,B 0,C 180,E1 -27866.503,E2 -27866.503} C_VEL
LIN {X 0,Y 125.638,Z 563.583,A -85,B 0,C 180,E1 -27868.546,E2 -27868.546} C_VEL
LIN {X 0,Y 130.611,Z 552.164,A -85,B 0,C 180,E1 -27870.188,E2 -27870.188} C_VEL
LIN {X 0,Y 134.684,Z 540.383,A -85,B 0,C 180,E1 -27871.318,E2 -27871.318} C_VEL
LIN {X 0,Y 137.841,Z 527.178,A -85,B 0,C 180,E1 -27872.274,E2 -27872.274} C_VEL
LIN {X 0,Y 139.601,Z 515.463,A -85,B 0,C 180,E1 -27872.821,E2 -27872.821} C_VEL
LIN {X 0,Y 140.962,Z 501.143,A -85,B 0,C 180,E1 -27873.339,E2 -27873.339} C_VEL
LIN {X 0,Y 138.828,Z 494.209,A -85,B 0,C 180,E1 -27875.977,E2 -27875.977} C_VEL
LIN {X 0,Y 137.841,Z 491.905,A -85,B 0,C 180,E1 -27877.206,E2 -27877.206} C_VEL
LIN {X 0,Y 136.036,Z 489.782,A -85,B 0,C 180,E1 -27879.377,E2 -27879.377} C_VEL
LIN {X 0,Y 132.985,Z 488.292,A -85,B 0,C 180,E1 -27883.439,E2 -27883.439} C_VEL
LIN {X 0,Y 131.005,Z 487.102,A -85,B 0,C 180,E1 -27886.885,E2 -27886.885} C_VEL
LIN {X 0,Y 130.301,Z 485.903,A -85,B 0,C 180,E1 -27888.583,E2 -27888.583} C_VEL
LIN {X 0,Y 129.621,Z 484.378,A -85,B 0,C 180,E1 -27890.639,E2 -27890.639} C_VEL
LIN {X 0,Y 128.35,Z 480.107,A -85,B 0,C 180,E1 -27900,E2 -27900} C_VEL
LIN {X 0,Y 128.351,Z 480.588,A -85,B 0,C 180,E1 -27901.961,E2 -27901.961} C_VEL
LIN {X 0,Y 129.957,Z 484.97,A -85,B 0,C 180,E1 -27910.759,E2 -27910.759} C_VEL
LIN {X 0,Y 131.764,Z 488.773,A -85,B 0,C 180,E1 -27915.17,E2 -27915.17} C_VEL
LIN {X 0,Y 133.837,Z 493.036,A -85,B 0,C 180,E1 -27918.902,E2 -27918.902} C_VEL
LIN {X 0,Y 136.433,Z 498.789,A -85,B 0,C 180,E1 -27922.68,E2 -27922.68} C_VEL
LIN {X 0,Y 137.771,Z 502.172,A -85,B 0,C 180,E1 -27924.413,E2 -27924.413} C_VEL
LIN {X 0,Y 135.667,Z 520.431,A -85,B 0,C 180,E1 -27925.14,E2 -27925.14} C_VEL
LIN {X 0,Y 132.858,Z 533.446,A -85,B 0,C 180,E1 -27925.937,E2 -27925.937} C_VEL
LIN {X 0,Y 129.178,Z 545.204,A -85,B 0,C 180,E1 -27927.015,E2 -27927.015} C_VEL
LIN {X 0,Y 124.852,Z 555.984,A -85,B 0,C 180,E1 -27928.413,E2 -27928.413} C_VEL
LIN {X 0,Y 119.138,Z 567.307,A -85,B 0,C 180,E1 -27930.375,E2 -27930.375} C_VEL
LIN {X 0,Y 112.885,Z 577.51,A -85,B 0,C 180,E1 -27932.809,E2 -27932.809} C_VEL
LIN {X 0,Y 106.193,Z 586.67,A -85,B 0,C 180,E1 -27935.834,E2 -27935.834} C_VEL
LIN {X 0,Y 98.733,Z 595.552,A -85,B 0,C 180,E1 -27940.055,E2 -27940.055} C_VEL
LIN {X 0,Y 91.786,Z 602.731,A -85,B 0,C 180,E1 -27944.907,E2 -27944.907} C_VEL
LIN {X 0,Y 86.372,Z 607.562,A -85,B 0,C 180,E1 -27949.388,E2 -27949.388} C_VEL
LIN {X 0,Y 80.725,Z 612.254,A -85,B 0,C 180,E1 -27955.536,E2 -27955.536} C_VEL
LIN {X 0,Y 76.162,Z 615.838,A -85,B 0,C 180,E1 -27962.525,E2 -27962.525} C_VEL
LIN {X 0,Y 73.777,Z 617.687,A -85,B 0,C 180,E1 -27967.603,E2 -27967.603} C_VEL
LIN {X 0,Y 71.884,Z 619.074,A -85,B 0,C 180,E1 -27972.945,E2 -27972.945} C_VEL
LIN {X 0,Y 69.921,Z 620.662,A -85,B 0,C 180,E1 -27984.232,E2 -27984.232} C_VEL
LIN {X 0,Y 69.75,Z 620.885,A -85,B 0,C 180,E1 -27990.001,E2 -27990.001} C_VEL
LIN {X 0,Y 69.921,Z 620.688,A -85,B 0,C 180,E1 -27995.77,E2 -27995.77} C_VEL
LIN {X 0,Y 71.884,Z 619.133,A -85,B 0,C 180,E1 -28007.057,E2 -28007.057} C_VEL
LIN {X 0,Y 73.774,Z 617.772,A -85,B 0,C 180,E1 -28012.4,E2 -28012.4} C_VEL
LIN {X 0,Y 77.541,Z 614.898,A -85,B 0,C 180,E1 -28019.902,E2 -28019.902} C_VEL
LIN {X 0,Y 82.412,Z 610.999,A -85,B 0,C 180,E1 -28026.653,E2 -28026.653} C_VEL
LIN {X 0,Y 88.423,Z 605.962,A -85,B 0,C 180,E1 -28032.502,E2 -28032.502} C_VEL
LIN {X 0,Y 95.062,Z 599.62,A -85,B 0,C 180,E1 -28037.674,E2 -28037.674} C_VEL
LIN {X 0,Y 102.299,Z 591.689,A -85,B 0,C 180,E1 -28042.192,E2 -28042.192} C_VEL
LIN {X 0,Y 108.749,Z 583.602,A -85,B 0,C 180,E1 -28045.487,E2 -28045.487} C_VEL
LIN {X 0,Y 115.595,Z 573.727,A -85,B 0,C 180,E1 -28048.342,E2 -28048.342} C_VEL
LIN {X 0,Y 121.907,Z 562.6,A -85,B 0,C 180,E1 -28050.69,E2 -28050.69} C_VEL
LIN {X 0,Y 126.947,Z 551.691,A -85,B 0,C 180,E1 -28052.351,E2 -28052.351} C_VEL
LIN {X 0,Y 131.339,Z 539.623,A -85,B 0,C 180,E1 -28053.678,E2 -28053.678} C_VEL
LIN {X 0,Y 134.751,Z 526.64,A -85,B 0,C 180,E1 -28054.669,E2 -28054.669} C_VEL
LIN {X 0,Y 136.915,Z 513.656,A -85,B 0,C 180,E1 -28055.283,E2 -28055.283} C_VEL
LIN {X 0,Y 138.07,Z 502.422,A -85,B 0,C 180,E1 -28055.67,E2 -28055.67} C_VEL
LIN {X 0,Y 135.556,Z 496.391,A -85,B 0,C 180,E1 -28059.019,E2 -28059.019} C_VEL
LIN {X 0,Y 133.002,Z 490.951,A -85,B 0,C 180,E1 -28063.104,E2 -28063.104} C_VEL
LIN {X 0,Y 131.257,Z 487.472,A -85,B 0,C 180,E1 -28066.649,E2 -28066.649} C_VEL
LIN {X 0,Y 129.955,Z 484.578,A -85,B 0,C 180,E1 -28070.27,E2 -28070.27} C_VEL
LIN {X 0,Y 128.643,Z 480.48,A -85,B 0,C 180,E1 -28080,E2 -28080} C_VEL
LIN {X 0,Y 130.15,Z 485.129,A -85,B 0,C 180,E1 -28090.108,E2 -28090.108} C_VEL
LIN {X 0,Y 132.026,Z 489.023,A -85,B 0,C 180,E1 -28094.745,E2 -28094.745} C_VEL
LIN {X 0,Y 134.067,Z 493.184,A -85,B 0,C 180,E1 -28098.431,E2 -28098.431} C_VEL
LIN {X 0,Y 135.967,Z 497.572,A -85,B 0,C 180,E1 -28101.312,E2 -28101.312} C_VEL
LIN {X 0,Y 137.863,Z 504.15,A -85,B 0,C 180,E1 -28104.068,E2 -28104.068} C_VEL
LIN {X 0,Y 136.059,Z 520.832,A -85,B 0,C 180,E1 -28104.712,E2 -28104.712} C_VEL
LIN {X 0,Y 133.238,Z 534.462,A -85,B 0,C 180,E1 -28105.434,E2 -28105.434} C_VEL
LIN {X 0,Y 129.522,Z 546.719,A -85,B 0,C 180,E1 -28106.45,E2 -28106.45} C_VEL
LIN {X 0,Y 124.324,Z 559.359,A -85,B 0,C 180,E1 -28107.958,E2 -28107.958} C_VEL
LIN {X 0,Y 118.456,Z 570.606,A -85,B 0,C 180,E1 -28109.805,E2 -28109.805} C_VEL
LIN {X 0,Y 112.13,Z 580.739,A -85,B 0,C 180,E1 -28112.203,E2 -28112.203} C_VEL
LIN {X 0,Y 105.32,Z 589.873,A -85,B 0,C 180,E1 -28115.168,E2 -28115.168} C_VEL
LIN {X 0,Y 97.625,Z 598.78,A -85,B 0,C 180,E1 -28119.294,E2 -28119.294} C_VEL
LIN {X 0,Y 90.14,Z 606.411,A -85,B 0,C 180,E1 -28124.564,E2 -28124.564} C_VEL
LIN {X 0,Y 85.412,Z 610.793,A -85,B 0,C 180,E1 -28128.831,E2 -28128.831} C_VEL
LIN {X 0,Y 79.786,Z 615.498,A -85,B 0,C 180,E1 -28135.07,E2 -28135.07} C_VEL
LIN {X 0,Y 75.19,Z 619.093,A -85,B 0,C 180,E1 -28142.136,E2 -28142.136} C_VEL
LIN {X 0,Y 72.942,Z 620.95,A -85,B 0,C 180,E1 -28147.33,E2 -28147.33} C_VEL
LIN {X 0,Y 70.145,Z 623.343,A -85,B 0,C 180,E1 -28158.439,E2 -28158.439} C_VEL
LIN {X 0,Y 69.62,Z 623.953,A -85,B 0,C 180,E1 -28164.205,E2 -28164.205} C_VEL
LIN {X 0,Y 69.644,Z 624.167,A -85,B 0,C 180,E1 -28169.999,E2 -28169.999} C_VEL
LIN {X 0,Y 69.62,Z 623.934,A -85,B 0,C 180,E1 -28175.793,E2 -28175.793} C_VEL
LIN {X 0,Y 70.145,Z 623.313,A -85,B 0,C 180,E1 -28181.558,E2 -28181.558} C_VEL
LIN {X 0,Y 71.235,Z 622.302,A -85,B 0,C 180,E1 -28187.215,E2 -28187.215} C_VEL
LIN {X 0,Y 72.94,Z 620.89,A -85,B 0,C 180,E1 -28192.668,E2 -28192.668} C_VEL
LIN {X 0,Y 76.598,Z 617.935,A -85,B 0,C 180,E1 -28200.306,E2 -28200.306} C_VEL
LIN {X 0,Y 81.521,Z 613.947,A -85,B 0,C 180,E1 -28207.118,E2 -28207.118} C_VEL
LIN {X 0,Y 87.463,Z 608.822,A -85,B 0,C 180,E1 -28213.079,E2 -28213.079} C_VEL
LIN {X 0,Y 93.989,Z 602.361,A -85,B 0,C 180,E1 -28218.395,E2 -28218.395} C_VEL
LIN {X 0,Y 101.398,Z 594.323,A -85,B 0,C 180,E1 -28222.851,E2 -28222.851} C_VEL
LIN {X 0,Y 107.984,Z 586.13,A -85,B 0,C 180,E1 -28226.079,E2 -28226.079} C_VEL
LIN {X 0,Y 114.888,Z 576.139,A -85,B 0,C 180,E1 -28228.916,E2 -28228.916} C_VEL
LIN {X 0,Y 120.636,Z 566.266,A -85,B 0,C 180,E1 -28230.91,E2 -28230.91} C_VEL
LIN {X 0,Y 126.497,Z 553.764,A -85,B 0,C 180,E1 -28232.739,E2 -28232.739} C_VEL
LIN {X 0,Y 130.658,Z 542.603,A -85,B 0,C 180,E1 -28233.845,E2 -28233.845} C_VEL
LIN {X 0,Y 134.119,Z 529.739,A -85,B 0,C 180,E1 -28234.802,E2 -28234.802} C_VEL
LIN {X 0,Y 136.281,Z 517.207,A -85,B 0,C 180,E1 -28235.393,E2 -28235.393} C_VEL
LIN {X 0,Y 137.622,Z 503.895,A -85,B 0,C 180,E1 -28235.887,E2 -28235.887} C_VEL
LIN {X 0,Y 135.481,Z 496.585,A -85,B 0,C 180,E1 -28239.004,E2 -28239.004} C_VEL
LIN {X 0,Y 132.888,Z 490.973,A -85,B 0,C 180,E1 -28243.09,E2 -28243.09} C_VEL
LIN {X 0,Y 131.033,Z 487.305,A -85,B 0,C 180,E1 -28246.786,E2 -28246.786} C_VEL
LIN {X 0,Y 130.301,Z 485.903,A -85,B 0,C 180,E1 -28248.583,E2 -28248.583} C_VEL
LIN {X 0,Y 129.759,Z 485.33,A -85,B 0,C 180,E1 -28249.987,E2 -28249.987} C_VEL
LIN {X 0,Y 128.934,Z 486.009,A -85,B 0,C 180,E1 -28252.014,E2 -28252.014} C_VEL
LIN {X 0,Y 127.647,Z 488.439,A -85,B 0,C 180,E1 -28256.122,E2 -28256.122} C_VEL
LIN {X 0,Y 127.456,Z 488.191,A -85,B 0,C 180,E1 -28257.923,E2 -28257.923} C_VEL
LIN {X 0,Y 127.479,Z 487.195,A -85,B 0,C 180,E1 -28260,E2 -28260} C_VEL
LIN {X 0,Y 127.464,Z 487.62,A -85,B 0,C 180,E1 -28261.58,E2 -28261.58} C_VEL
LIN {X 0,Y 128.765,Z 491.752,A -85,B 0,C 180,E1 -28269.902,E2 -28269.902} C_VEL
LIN {X 0,Y 130.368,Z 495.432,A -85,B 0,C 180,E1 -28274.239,E2 -28274.239} C_VEL
LIN {X 0,Y 132.399,Z 499.947,A -85,B 0,C 180,E1 -28278.197,E2 -28278.197} C_VEL
LIN {X 0,Y 134.643,Z 505.588,A -85,B 0,C 180,E1 -28281.751,E2 -28281.751} C_VEL
LIN {X 0,Y 132.64,Z 521.64,A -85,B 0,C 180,E1 -28282.416,E2 -28282.416} C_VEL
LIN {X 0,Y 129.91,Z 533.622,A -85,B 0,C 180,E1 -28283.121,E2 -28283.121} C_VEL
LIN {X 0,Y 126.055,Z 545.554,A -85,B 0,C 180,E1 -28284.17,E2 -28284.17} C_VEL
LIN {X 0,Y 121.639,Z 556.156,A -85,B 0,C 180,E1 -28285.476,E2 -28285.476} C_VEL
LIN {X 0,Y 115.709,Z 567.479,A -85,B 0,C 180,E1 -28287.341,E2 -28287.341} C_VEL
LIN {X 0,Y 109.202,Z 577.681,A -85,B 0,C 180,E1 -28289.678,E2 -28289.678} C_VEL
LIN {X 0,Y 102.198,Z 586.839,A -85,B 0,C 180,E1 -28292.605,E2 -28292.605} C_VEL
LIN {X 0,Y 95.378,Z 594.592,A -85,B 0,C 180,E1 -28296.121,E2 -28296.121} C_VEL
LIN {X 0,Y 88.089,Z 601.79,A -85,B 0,C 180,E1 -28300.719,E2 -28300.719} C_VEL
LIN {X 0,Y 81.111,Z 607.731,A -85,B 0,C 180,E1 -28306.119,E2 -28306.119} C_VEL
LIN {X 0,Y 74.969,Z 612.422,A -85,B 0,C 180,E1 -28312.459,E2 -28312.459} C_VEL
LIN {X 0,Y 69.933,Z 616.006,A -85,B 0,C 180,E1 -28319.837,E2 -28319.837} C_VEL
LIN {X 0,Y 67.273,Z 617.854,A -85,B 0,C 180,E1 -28325.3,E2 -28325.3} C_VEL
LIN {X 0,Y 63.655,Z 620.227,A -85,B 0,C 180,E1 -28337.244,E2 -28337.244} C_VEL
LIN {X 0,Y 62.879,Z 620.829,A -85,B 0,C 180,E1 -28343.584,E2 -28343.584} C_VEL
LIN {X 0,Y 62.676,Z 621.052,A -85,B 0,C 180,E1 -28350.001,E2 -28350.001} C_VEL
LIN {X 0,Y 62.879,Z 620.855,A -85,B 0,C 180,E1 -28356.419,E2 -28356.419} C_VEL
LIN {X 0,Y 65.119,Z 619.3,A -85,B 0,C 180,E1 -28368.893,E2 -28368.893} C_VEL
LIN {X 0,Y 67.269,Z 617.938,A -85,B 0,C 180,E1 -28374.704,E2 -28374.704} C_VEL
LIN {X 0,Y 71.468,Z 615.064,A -85,B 0,C 180,E1 -28382.743,E2 -28382.743} C_VEL
LIN {X 0,Y 76.834,Z 611.165,A -85,B 0,C 180,E1 -28389.815,E2 -28389.815} C_VEL
LIN {X 0,Y 83.327,Z 606.127,A -85,B 0,C 180,E1 -28395.801,E2 -28395.801} C_VEL
LIN {X 0,Y 90.438,Z 599.785,A -85,B 0,C 180,E1 -28400.998,E2 -28400.998} C_VEL
LIN {X 0,Y 98.106,Z 591.854,A -85,B 0,C 180,E1 -28405.471,E2 -28405.471} C_VEL
LIN {X 0,Y 104.895,Z 583.766,A -85,B 0,C 180,E1 -28408.679,E2 -28408.679} C_VEL
LIN {X 0,Y 112.034,Z 573.891,A -85,B 0,C 180,E1 -28411.432,E2 -28411.432} C_VEL
LIN {X 0,Y 118.598,Z 562.762,A -85,B 0,C 180,E1 -28413.677,E2 -28413.677} C_VEL
LIN {X 0,Y 123.82,Z 551.852,A -85,B 0,C 180,E1 -28415.254,E2 -28415.254} C_VEL
LIN {X 0,Y 128.352,Z 539.782,A -85,B 0,C 180,E1 -28416.516,E2 -28416.516} C_VEL
LIN {X 0,Y 131.795,Z 527.189,A -85,B 0,C 180,E1 -28417.428,E2 -28417.428} C_VEL
LIN {X 0,Y 134.053,Z 514.201,A -85,B 0,C 180,E1 -28418.024,E2 -28418.024} C_VEL
LIN {X 0,Y 134.951,Z 505.905,A -85,B 0,C 180,E1 -28418.311,E2 -28418.311} C_VEL
LIN {X 0,Y 132.649,Z 500.109,A -85,B 0,C 180,E1 -28421.964,E2 -28421.964} C_VEL
LIN {X 0,Y 130.803,Z 496.105,A -85,B 0,C 180,E1 -28425.512,E2 -28425.512} C_VEL
LIN {X 0,Y 129.815,Z 493.91,A -85,B 0,C 180,E1 -28427.89,E2 -28427.89} C_VEL
LIN {X 0,Y 128.701,Z 491.238,A -85,B 0,C 180,E1 -28431.462,E2 -28431.462} C_VEL
LIN {X 0,Y 127.755,Z 487.712,A -85,B 0,C 180,E1 -28440,E2 -28440} C_VEL
LIN {X 0,Y 128.964,Z 491.835,A -85,B 0,C 180,E1 -28449.212,E2 -28449.212} C_VEL
LIN {X 0,Y 130.569,Z 495.55,A -85,B 0,C 180,E1 -28453.67,E2 -28453.67} C_VEL
LIN {X 0,Y 132.461,Z 499.738,A -85,B 0,C 180,E1 -28457.431,E2 -28457.431} C_VEL
LIN {X 0,Y 133.835,Z 503.291,A -85,B 0,C 180,E1 -28459.758,E2 -28459.758} C_VEL
LIN {X 0,Y 134.807,Z 507.003,A -85,B 0,C 180,E1 -28461.404,E2 -28461.404} C_VEL
LIN {X 0,Y 133.175,Z 521.111,A -85,B 0,C 180,E1 -28461.956,E2 -28461.956} C_VEL
LIN {X 0,Y 130.394,Z 534.121,A -85,B 0,C 180,E1 -28462.604,E2 -28462.604} C_VEL
LIN {X 0,Y 126.524,Z 546.559,A -85,B 0,C 180,E1 -28463.575,E2 -28463.575} C_VEL
LIN {X 0,Y 121.163,Z 559.197,A -85,B 0,C 180,E1 -28464.996,E2 -28464.996} C_VEL
LIN {X 0,Y 115.095,Z 570.443,A -85,B 0,C 180,E1 -28466.74,E2 -28466.74} C_VEL
LIN {X 0,Y 108.497,Z 580.574,A -85,B 0,C 180,E1 -28469.015,E2 -28469.015} C_VEL
LIN {X 0,Y 101.395,Z 589.708,A -85,B 0,C 180,E1 -28471.886,E2 -28471.886} C_VEL
LIN {X 0,Y 93.276,Z 598.614,A -85,B 0,C 180,E1 -28475.905,E2 -28475.905} C_VEL
LIN {X 0,Y 86.764,Z 604.893,A -85,B 0,C 180,E1 -28480.05,E2 -28480.05} C_VEL
LIN {X 0,Y 80.195,Z 610.627,A -85,B 0,C 180,E1 -28485.484,E2 -28485.484} C_VEL
LIN {X 0,Y 74.06,Z 615.331,A -85,B 0,C 180,E1 -28491.914,E2 -28491.914} C_VEL
LIN {X 0,Y 68.97,Z 618.926,A -85,B 0,C 180,E1 -28499.368,E2 -28499.368} C_VEL
LIN {X 0,Y 66.403,Z 620.783,A -85,B 0,C 180,E1 -28504.952,E2 -28504.952} C_VEL
LIN {X 0,Y 64.473,Z 622.177,A -85,B 0,C 180,E1 -28510.91,E2 -28510.91} C_VEL
LIN {X 0,Y 62.555,Z 623.786,A -85,B 0,C 180,E1 -28523.548,E2 -28523.548} C_VEL
LIN {X 0,Y 62.544,Z 624,A -85,B 0,C 180,E1 -28529.999,E2 -28529.999} C_VEL
LIN {X 0,Y 62.555,Z 623.767,A -85,B 0,C 180,E1 -28536.45,E2 -28536.45} C_VEL
LIN {X 0,Y 64.471,Z 622.134,A -85,B 0,C 180,E1 -28549.087,E2 -28549.087} C_VEL
LIN {X 0,Y 66.4,Z 620.721,A -85,B 0,C 180,E1 -28555.046,E2 -28555.046} C_VEL
LIN {X 0,Y 70.543,Z 617.767,A -85,B 0,C 180,E1 -28563.226,E2 -28563.226} C_VEL
LIN {X 0,Y 75.95,Z 613.778,A -85,B 0,C 180,E1 -28570.371,E2 -28570.371} C_VEL
LIN {X 0,Y 81.785,Z 609.155,A -85,B 0,C 180,E1 -28575.946,E2 -28575.946} C_VEL
LIN {X 0,Y 89.417,Z 602.191,A -85,B 0,C 180,E1 -28581.811,E2 -28581.811} C_VEL
LIN {X 0,Y 97.271,Z 594.153,A -85,B 0,C 180,E1 -28586.19,E2 -28586.19} C_VEL
LIN {X 0,Y 104.189,Z 585.96,A -85,B 0,C 180,E1 -28589.321,E2 -28589.321} C_VEL
LIN {X 0,Y 111.39,Z 575.968,A -85,B 0,C 180,E1 -28592.044,E2 -28592.044} C_VEL
LIN {X 0,Y 117.346,Z 566.094,A -85,B 0,C 180,E1 -28593.944,E2 -28593.944} C_VEL
LIN {X 0,Y 123.412,Z 553.592,A -85,B 0,C 180,E1 -28595.665,E2 -28595.665} C_VEL
LIN {X 0,Y 127.686,Z 542.45,A -85,B 0,C 180,E1 -28596.698,E2 -28596.698} C_VEL
LIN {X 0,Y 131.275,Z 529.484,A -85,B 0,C 180,E1 -28597.606,E2 -28597.606} C_VEL
LIN {X 0,Y 133.553,Z 516.386,A -85,B 0,C 180,E1 -28598.195,E2 -28598.195} C_VEL
LIN {X 0,Y 134.558,Z 506.73,A -85,B 0,C 180,E1 -28598.555,E2 -28598.555} C_VEL
LIN {X 0,Y 133.181,Z 501.882,A -85,B 0,C 180,E1 -28600.861,E2 -28600.861} C_VEL
LIN {X 0,Y 131.062,Z 496.94,A -85,B 0,C 180,E1 -28604.667,E2 -28604.667} C_VEL
LIN {X 0,Y 129.569,Z 493.702,A -85,B 0,C 180,E1 -28608.065,E2 -28608.065} C_VEL
LIN {X 0,Y 128.509,Z 491.227,A -85,B 0,C 180,E1 -28611.35,E2 -28611.35} C_VEL
LIN {X 0,Y 127.456,Z 488.191,A -85,B 0,C 180,E1 -28617.923,E2 -28617.923} C_VEL
LIN {X 0,Y 127.372,Z 488.176,A -85,B 0,C 180,E1 -28619.343,E2 -28619.343} C_VEL
LIN {X 0,Y 127.156,Z 489.997,A -85,B 0,C 180,E1 -28621.236,E2 -28621.236} C_VEL
LIN {X 0,Y 126.844,Z 495.759,A -85,B 0,C 180,E1 -28624.833,E2 -28624.833} C_VEL
LIN {X 0,Y 127.025,Z 497.337,A -85,B 0,C 180,E1 -28626.591,E2 -28626.591} C_VEL
LIN {X 0,Y 127.677,Z 498.719,A -85,B 0,C 180,E1 -28629.306,E2 -28629.306} C_VEL
LIN {X 0,Y 128.995,Z 502.078,A -85,B 0,C 180,E1 -28633.263,E2 -28633.263} C_VEL
LIN {X 0,Y 130.623,Z 506.039,A -85,B 0,C 180,E1 -28636.81,E2 -28636.81} C_VEL
LIN {X 0,Y 131.809,Z 509.288,A -85,B 0,C 180,E1 -28639.003,E2 -28639.003} C_VEL
LIN {X 0,Y 129.982,Z 522.521,A -85,B 0,C 180,E1 -28639.567,E2 -28639.567} C_VEL
LIN {X 0,Y 127.291,Z 533.797,A -85,B 0,C 180,E1 -28640.182,E2 -28640.182} C_VEL
LIN {X 0,Y 123.177,Z 546.099,A -85,B 0,C 180,E1 -28641.201,E2 -28641.201} C_VEL
LIN {X 0,Y 118,Z 557.906,A -85,B 0,C 180,E1 -28642.606,E2 -28642.606} C_VEL
LIN {X 0,Y 111.877,Z 568.924,A -85,B 0,C 180,E1 -28644.374,E2 -28644.374} C_VEL
LIN {X 0,Y 105.869,Z 577.851,A -85,B 0,C 180,E1 -28646.34,E2 -28646.34} C_VEL
LIN {X 0,Y 98.56,Z 587.009,A -85,B 0,C 180,E1 -28649.132,E2 -28649.132} C_VEL
LIN {X 0,Y 90.956,Z 595.176,A -85,B 0,C 180,E1 -28652.744,E2 -28652.744} C_VEL
LIN {X 0,Y 83.611,Z 601.96,A -85,B 0,C 180,E1 -28657.011,E2 -28657.011} C_VEL
LIN {X 0,Y 76.154,Z 607.899,A -85,B 0,C 180,E1 -28662.415,E2 -28662.415} C_VEL
LIN {X 0,Y 69.47,Z 612.591,A -85,B 0,C 180,E1 -28668.886,E2 -28668.886} C_VEL
LIN {X 0,Y 63.894,Z 616.174,A -85,B 0,C 180,E1 -28676.636,E2 -28676.636} C_VEL
LIN {X 0,Y 60.878,Z 618.023,A -85,B 0,C 180,E1 -28682.499,E2 -28682.499} C_VEL
LIN {X 0,Y 56.755,Z 620.395,A -85,B 0,C 180,E1 -28695.662,E2 -28695.662} C_VEL
LIN {X 0,Y 55.83,Z 620.997,A -85,B 0,C 180,E1 -28702.77,E2 -28702.77} C_VEL
LIN {X 0,Y 55.592,Z 621.219,A -85,B 0,C 180,E1 -28710.001,E2 -28710.001} C_VEL
LIN {X 0,Y 55.831,Z 621.022,A -85,B 0,C 180,E1 -28717.233,E2 -28717.233} C_VEL
LIN {X 0,Y 58.447,Z 619.467,A -85,B 0,C 180,E1 -28731.147,E2 -28731.147} C_VEL
LIN {X 0,Y 60.874,Z 618.105,A -85,B 0,C 180,E1 -28737.506,E2 -28737.506} C_VEL
LIN {X 0,Y 65.606,Z 615.231,A -85,B 0,C 180,E1 -28746.101,E2 -28746.101} C_VEL
LIN {X 0,Y 71.529,Z 611.331,A -85,B 0,C 180,E1 -28753.456,E2 -28753.456} C_VEL
LIN {X 0,Y 78.544,Z 606.293,A -85,B 0,C 180,E1 -28759.516,E2 -28759.516} C_VEL
LIN {X 0,Y 86.152,Z 599.95,A -85,B 0,C 180,E1 -28764.665,E2 -28764.665} C_VEL
LIN {X 0,Y 94.256,Z 592.019,A -85,B 0,C 180,E1 -28769.036,E2 -28769.036} C_VEL
LIN {X 0,Y 101.391,Z 583.93,A -85,B 0,C 180,E1 -28772.103,E2 -28772.103} C_VEL
LIN {X 0,Y 108.809,Z 574.055,A -85,B 0,C 180,E1 -28774.727,E2 -28774.727} C_VEL
LIN {X 0,Y 115.63,Z 562.924,A -85,B 0,C 180,E1 -28776.826,E2 -28776.826} C_VEL
LIN {X 0,Y 121.029,Z 552.013,A -85,B 0,C 180,E1 -28778.298,E2 -28778.298} C_VEL
LIN {X 0,Y 125.492,Z 540.542,A -85,B 0,C 180,E1 -28779.425,E2 -28779.425} C_VEL
LIN {X 0,Y 129.159,Z 527.708,A -85,B 0,C 180,E1 -28780.315,E2 -28780.315} C_VEL
LIN {X 0,Y 131.472,Z 515.096,A -85,B 0,C 180,E1 -28780.86,E2 -28780.86} C_VEL
LIN {X 0,Y 132.102,Z 509.507,A -85,B 0,C 180,E1 -28781.09,E2 -28781.09} C_VEL
LIN {X 0,Y 130.026,Z 504.04,A -85,B 0,C 180,E1 -28785.123,E2 -28785.123} C_VEL
LIN {X 0,Y 128.676,Z 500.803,A -85,B 0,C 180,E1 -28788.481,E2 -28788.481} C_VEL
LIN {X 0,Y 127.65,Z 498.107,A -85,B 0,C 180,E1 -28792.088,E2 -28792.088} C_VEL
LIN {X 0,Y 126.871,Z 494.917,A -85,B 0,C 180,E1 -28800,E2 -28800} C_VEL
LIN {X 0,Y 127.883,Z 498.806,A -85,B 0,C 180,E1 -28808.613,E2 -28808.613} C_VEL
LIN {X 0,Y 129.233,Z 502.269,A -85,B 0,C 180,E1 -28812.763,E2 -28812.763} C_VEL
LIN {X 0,Y 130.698,Z 505.793,A -85,B 0,C 180,E1 -28816.014,E2 -28816.014} C_VEL
LIN {X 0,Y 131.856,Z 509.221,A -85,B 0,C 180,E1 -28818.257,E2 -28818.257} C_VEL
LIN {X 0,Y 132.069,Z 510.13,A -85,B 0,C 180,E1 -28818.685,E2 -28818.685} C_VEL
LIN {X 0,Y 130.055,Z 524.533,A -85,B 0,C 180,E1 -28819.2,E2 -28819.2} C_VEL
LIN {X 0,Y 127.013,Z 536.857,A -85,B 0,C 180,E1 -28819.834,E2 -28819.834} C_VEL
LIN {X 0,Y 123.022,Z 548.52,A -85,B 0,C 180,E1 -28820.766,E2 -28820.766} C_VEL
LIN {X 0,Y 117.551,Z 560.618,A -85,B 0,C 180,E1 -28822.072,E2 -28822.072} C_VEL
LIN {X 0,Y 111.306,Z 571.522,A -85,B 0,C 180,E1 -28823.713,E2 -28823.713} C_VEL
LIN {X 0,Y 103.736,Z 582.365,A -85,B 0,C 180,E1 -28826.144,E2 -28826.144} C_VEL
LIN {X 0,Y 96.372,Z 591.174,A -85,B 0,C 180,E1 -28828.94,E2 -28828.94} C_VEL
LIN {X 0,Y 87.914,Z 599.76,A -85,B 0,C 180,E1 -28832.923,E2 -28832.923} C_VEL
LIN {X 0,Y 79.588,Z 607.034,A -85,B 0,C 180,E1 -28838.18,E2 -28838.18} C_VEL
LIN {X 0,Y 72.928,Z 612.147,A -85,B 0,C 180,E1 -28843.714,E2 -28843.714} C_VEL
LIN {X 0,Y 66.586,Z 616.469,A -85,B 0,C 180,E1 -28850.705,E2 -28850.705} C_VEL
LIN {X 0,Y 62.947,Z 618.759,A -85,B 0,C 180,E1 -28856.064,E2 -28856.064} C_VEL
LIN {X 0,Y 60.005,Z 620.615,A -85,B 0,C 180,E1 -28862.062,E2 -28862.062} C_VEL
LIN {X 0,Y 57.783,Z 622.01,A -85,B 0,C 180,E1 -28868.598,E2 -28868.598} C_VEL
LIN {X 0,Y 55.513,Z 623.619,A -85,B 0,C 180,E1 -28882.725,E2 -28882.725} C_VEL
LIN {X 0,Y 55.461,Z 623.833,A -85,B 0,C 180,E1 -28889.999,E2 -28889.999} C_VEL
LIN {X 0,Y 55.513,Z 623.6,A -85,B 0,C 180,E1 -28897.272,E2 -28897.272} C_VEL
LIN {X 0,Y 57.782,Z 621.966,A -85,B 0,C 180,E1 -28911.399,E2 -28911.399} C_VEL
LIN {X 0,Y 60.003,Z 620.552,A -85,B 0,C 180,E1 -28917.937,E2 -28917.937} C_VEL
LIN {X 0,Y 64.708,Z 617.599,A -85,B 0,C 180,E1 -28926.68,E2 -28926.68} C_VEL
LIN {X 0,Y 70.668,Z 613.609,A -85,B 0,C 180,E1 -28934.118,E2 -28934.118} C_VEL
LIN {X 0,Y 78.057,Z 608.102,A -85,B 0,C 180,E1 -28940.706,E2 -28940.706} C_VEL
LIN {X 0,Y 85.193,Z 602.022,A -85,B 0,C 180,E1 -28945.582,E2 -28945.582} C_VEL
LIN {X 0,Y 93.492,Z 593.983,A -85,B 0,C 180,E1 -28949.823,E2 -28949.823} C_VEL
LIN {X 0,Y 100.751,Z 585.79,A -85,B 0,C 180,E1 -28952.796,E2 -28952.796} C_VEL
LIN {X 0,Y 108.246,Z 575.798,A -85,B 0,C 180,E1 -28955.362,E2 -28955.362} C_VEL
LIN {X 0,Y 114.404,Z 565.923,A -85,B 0,C 180,E1 -28957.141,E2 -28957.141} C_VEL
LIN {X 0,Y 120.659,Z 553.419,A -85,B 0,C 180,E1 -28958.74,E2 -28958.74} C_VEL
LIN {X 0,Y 125.18,Z 541.927,A -85,B 0,C 180,E1 -28959.702,E2 -28959.702} C_VEL
LIN {X 0,Y 128.667,Z 529.649,A -85,B 0,C 180,E1 -28960.507,E2 -28960.507} C_VEL
LIN {X 0,Y 130.959,Z 517.186,A -85,B 0,C 180,E1 -28961.039,E2 -28961.039} C_VEL
LIN {X 0,Y 131.766,Z 509.841,A -85,B 0,C 180,E1 -28961.336,E2 -28961.336} C_VEL
LIN {X 0,Y 130.994,Z 507.104,A -85,B 0,C 180,E1 -28962.838,E2 -28962.838} C_VEL
LIN {X 0,Y 129.366,Z 502.968,A -85,B 0,C 180,E1 -28966.222,E2 -28966.222} C_VEL
LIN {X 0,Y 128.11,Z 499.888,A -85,B 0,C 180,E1 -28969.58,E2 -28969.58} C_VEL
LIN {X 0,Y 127.369,Z 497.973,A -85,B 0,C 180,E1 -28972.271,E2 -28972.271} C_VEL
LIN {X 0,Y 126.599,Z 494.365,A -85,B 0,C 180,E1 -28980,E2 -28980} C_VEL
LIN {X 0,Y 126.57,Z 494.889,A -85,B 0,C 180,E1 -28981.566,E2 -28981.566} C_VEL
LIN {X 0,Y 127.025,Z 497.337,A -85,B 0,C 180,E1 -28986.591,E2 -28986.591} C_VEL
LIN {X 0,Y 127.298,Z 498.822,A -85,B 0,C 180,E1 -28988.216,E2 -28988.216} C_VEL
LIN {X 0,Y 127.529,Z 502.172,A -85,B 0,C 180,E1 -28990.064,E2 -28990.064} C_VEL
LIN {X 0,Y 128.034,Z 508.97,A -85,B 0,C 180,E1 -28993.084,E2 -28993.084} C_VEL
LIN {X 0,Y 128.364,Z 510.535,A -85,B 0,C 180,E1 -28994.074,E2 -28994.074} C_VEL
LIN {X 0,Y 129.23,Z 513.139,A -85,B 0,C 180,E1 -28996.129,E2 -28996.129} C_VEL
LIN {X 0,Y 127.124,Z 525.657,A -85,B 0,C 180,E1 -28996.686,E2 -28996.686} C_VEL
LIN {X 0,Y 123.577,Z 538.697,A -85,B 0,C 180,E1 -28997.471,E2 -28997.471} C_VEL
LIN {X 0,Y 119.292,Z 549.949,A -85,B 0,C 180,E1 -28998.409,E2 -28998.409} C_VEL
LIN {X 0,Y 113.864,Z 561.068,A -85,B 0,C 180,E1 -28999.735,E2 -28999.735} C_VEL
LIN {X 0,Y 106.794,Z 572.616,A -85,B 0,C 180,E1 -29001.636,E2 -29001.636} C_VEL
LIN {X 0,Y 99.847,Z 581.919,A -85,B 0,C 180,E1 -29003.79,E2 -29003.79} C_VEL
LIN {X 0,Y 92.324,Z 590.39,A -85,B 0,C 180,E1 -29006.563,E2 -29006.563} C_VEL
LIN {X 0,Y 83.719,Z 598.625,A -85,B 0,C 180,E1 -29010.628,E2 -29010.628} C_VEL
LIN {X 0,Y 76.823,Z 604.263,A -85,B 0,C 180,E1 -29014.58,E2 -29014.58} C_VEL
LIN {X 0,Y 69.05,Z 609.757,A -85,B 0,C 180,E1 -29020.24,E2 -29020.24} C_VEL
LIN {X 0,Y 62.073,Z 614.066,A -85,B 0,C 180,E1 -29027.21,E2 -29027.21} C_VEL
LIN {X 0,Y 58.099,Z 616.342,A -85,B 0,C 180,E1 -29032.785,E2 -29032.785} C_VEL
LIN {X 0,Y 54.671,Z 618.191,A -85,B 0,C 180,E1 -29039.057,E2 -29039.057} C_VEL
LIN {X 0,Y 51.896,Z 619.577,A -85,B 0,C 180,E1 -29046.031,E2 -29046.031} C_VEL
LIN {X 0,Y 48.812,Z 621.164,A -85,B 0,C 180,E1 -29061.723,E2 -29061.723} C_VEL
LIN {X 0,Y 48.497,Z 621.386,A -85,B 0,C 180,E1 -29070.002,E2 -29070.002} C_VEL
LIN {X 0,Y 48.812,Z 621.188,A -85,B 0,C 180,E1 -29078.28,E2 -29078.28} C_VEL
LIN {X 0,Y 51.896,Z 619.633,A -85,B 0,C 180,E1 -29093.973,E2 -29093.973} C_VEL
LIN {X 0,Y 54.666,Z 618.272,A -85,B 0,C 180,E1 -29100.949,E2 -29100.949} C_VEL
LIN {X 0,Y 59.992,Z 615.398,A -85,B 0,C 180,E1 -29110.116,E2 -29110.116} C_VEL
LIN {X 0,Y 66.561,Z 611.496,A -85,B 0,C 180,E1 -29117.657,E2 -29117.657} C_VEL
LIN {X 0,Y 74.133,Z 606.459,A -85,B 0,C 180,E1 -29123.692,E2 -29123.692} C_VEL
LIN {X 0,Y 82.256,Z 600.115,A -85,B 0,C 180,E1 -29128.697,E2 -29128.697} C_VEL
LIN {X 0,Y 90.797,Z 592.185,A -85,B 0,C 180,E1 -29132.893,E2 -29132.893} C_VEL
LIN {X 0,Y 98.265,Z 584.094,A -85,B 0,C 180,E1 -29135.771,E2 -29135.771} C_VEL
LIN {X 0,Y 105.976,Z 574.218,A -85,B 0,C 180,E1 -29138.195,E2 -29138.195} C_VEL
LIN {X 0,Y 113.028,Z 563.087,A -85,B 0,C 180,E1 -29140.132,E2 -29140.132} C_VEL
LIN {X 0,Y 118.592,Z 552.174,A -85,B 0,C 180,E1 -29141.48,E2 -29141.48} C_VEL
LIN {X 0,Y 123.347,Z 540.233,A -85,B 0,C 180,E1 -29142.549,E2 -29142.549} C_VEL
LIN {X 0,Y 127.114,Z 527.072,A -85,B 0,C 180,E1 -29143.379,E2 -29143.379} C_VEL
LIN {X 0,Y 129.397,Z 514.652,A -85,B 0,C 180,E1 -29143.85,E2 -29143.85} C_VEL
LIN {X 0,Y 129.476,Z 513.33,A -85,B 0,C 180,E1 -29144.039,E2 -29144.039} C_VEL
LIN {X 0,Y 128.064,Z 509.278,A -85,B 0,C 180,E1 -29147.521,E2 -29147.521} C_VEL
LIN {X 0,Y 127.076,Z 506.574,A -85,B 0,C 180,E1 -29150.65,E2 -29150.65} C_VEL
LIN {X 0,Y 126.589,Z 504.967,A -85,B 0,C 180,E1 -29152.824,E2 -29152.824} C_VEL
LIN {X 0,Y 125.983,Z 502.2,A -85,B 0,C 180,E1 -29159.257,E2 -29159.257} C_VEL
LIN {X 0,Y 125.976,Z 502.248,A -85,B 0,C 180,E1 -29160.381,E2 -29160.381} C_VEL
LIN {X 0,Y 126.779,Z 505.584,A -85,B 0,C 180,E1 -29167.806,E2 -29167.806} C_VEL
LIN {X 0,Y 127.95,Z 509.007,A -85,B 0,C 180,E1 -29171.887,E2 -29171.887} C_VEL
LIN {X 0,Y 129.28,Z 512.656,A -85,B 0,C 180,E1 -29175.166,E2 -29175.166} C_VEL
LIN {X 0,Y 129.582,Z 513.619,A -85,B 0,C 180,E1 -29175.845,E2 -29175.845} C_VEL
LIN {X 0,Y 127.279,Z 527.228,A -85,B 0,C 180,E1 -29176.33,E2 -29176.33} C_VEL
LIN {X 0,Y 123.73,Z 540.065,A -85,B 0,C 180,E1 -29176.971,E2 -29176.971} C_VEL
LIN {X 0,Y 119.054,Z 552.257,A -85,B 0,C 180,E1 -29177.962,E2 -29177.962} C_VEL
LIN {X 0,Y 112.659,Z 564.821,A -85,B 0,C 180,E1 -29179.341,E2 -29179.341} C_VEL
LIN {X 0,Y 105.491,Z 576.004,A -85,B 0,C 180,E1 -29181.137,E2 -29181.137} C_VEL
LIN {X 0,Y 97.717,Z 585.93,A -85,B 0,C 180,E1 -29183.505,E2 -29183.505} C_VEL
LIN {X 0,Y 90.121,Z 594.07,A -85,B 0,C 180,E1 -29186.254,E2 -29186.254} C_VEL
LIN {X 0,Y 81.399,Z 602.065,A -85,B 0,C 180,E1 -29190.297,E2 -29190.297} C_VEL
LIN {X 0,Y 73.312,Z 608.439,A -85,B 0,C 180,E1 -29195.339,E2 -29195.339} C_VEL
LIN {X 0,Y 65.747,Z 613.565,A -85,B 0,C 180,E1 -29201.558,E2 -29201.558} C_VEL
LIN {X 0,Y 59.162,Z 617.522,A -85,B 0,C 180,E1 -29209.202,E2 -29209.202} C_VEL
LIN {X 0,Y 53.798,Z 620.448,A -85,B 0,C 180,E1 -29218.495,E2 -29218.495} C_VEL
LIN {X 0,Y 49.397,Z 622.841,A -85,B 0,C 180,E1 -29233.466,E2 -29233.466} C_VEL
LIN {X 0,Y 48.474,Z 623.452,A -85,B 0,C 180,E1 -29241.662,E2 -29241.662} C_VEL
LIN {X 0,Y 48.362,Z 623.666,A -85,B 0,C 180,E1 -29249.998,E2 -29249.998} C_VEL
LIN {X 0,Y 48.474,Z 623.432,A -85,B 0,C 180,E1 -29258.335,E2 -29258.335} C_VEL
LIN {X 0,Y 51.197,Z 621.798,A -85,B 0,C 180,E1 -29274.318,E2 -29274.318} C_VEL
LIN {X 0,Y 53.796,Z 620.383,A -85,B 0,C 180,E1 -29281.503,E2 -29281.503} C_VEL
LIN {X 0,Y 59.158,Z 617.43,A -85,B 0,C 180,E1 -29290.797,E2 -29290.797} C_VEL
LIN {X 0,Y 65.742,Z 613.44,A -85,B 0,C 180,E1 -29298.444,E2 -29298.444} C_VEL
LIN {X 0,Y 73.046,Z 608.45,A -85,B 0,C 180,E1 -29304.513,E2 -29304.513} C_VEL
LIN {X 0,Y 81.386,Z 601.852,A -85,B 0,C 180,E1 -29309.715,E2 -29309.715} C_VEL
LIN {X 0,Y 90.115,Z 593.812,A -85,B 0,C 180,E1 -29313.75,E2 -29313.75} C_VEL
LIN {X 0,Y 97.708,Z 585.62,A -85,B 0,C 180,E1 -29316.503,E2 -29316.503} C_VEL
LIN {X 0,Y 105.486,Z 575.628,A -85,B 0,C 180,E1 -29318.866,E2 -29318.866} C_VEL
LIN {X 0,Y 112.642,Z 564.324,A -85,B 0,C 180,E1 -29320.678,E2 -29320.678} C_VEL
LIN {X 0,Y 118.27,Z 553.246,A -85,B 0,C 180,E1 -29321.946,E2 -29321.946} C_VEL
LIN {X 0,Y 123.035,Z 541.375,A -85,B 0,C 180,E1 -29322.832,E2 -29322.832} C_VEL
LIN {X 0,Y 126.679,Z 528.529,A -85,B 0,C 180,E1 -29323.59,E2 -29323.59} C_VEL
LIN {X 0,Y 128.975,Z 515.861,A -85,B 0,C 180,E1 -29324.066,E2 -29324.066} C_VEL
LIN {X 0,Y 129.266,Z 513.227,A -85,B 0,C 180,E1 -29324.226,E2 -29324.226} C_VEL
LIN {X 0,Y 127.885,Z 509.309,A -85,B 0,C 180,E1 -29327.503,E2 -29327.503} C_VEL
LIN {X 0,Y 126.812,Z 506.361,A -85,B 0,C 180,E1 -29330.832,E2 -29330.832} C_VEL
LIN {X 0,Y 126.353,Z 504.883,A -85,B 0,C 180,E1 -29332.811,E2 -29332.811} C_VEL
LIN {X 0,Y 125.714,Z 501.569,A -85,B 0,C 180,E1 -29340,E2 -29340} C_VEL
LIN {X 0,Y 126.49,Z 505.263,A -85,B 0,C 180,E1 -29348.186,E2 -29348.186} C_VEL
LIN {X 0,Y 127.684,Z 508.727,A -85,B 0,C 180,E1 -29352.315,E2 -29352.315} C_VEL
LIN {X 0,Y 128.364,Z 510.535,A -85,B 0,C 180,E1 -29354.074,E2 -29354.074} C_VEL
LIN {X 0,Y 128.499,Z 512.299,A -85,B 0,C 180,E1 -29354.726,E2 -29354.726} C_VEL
LIN {X 0,Y 128.213,Z 515.267,A -85,B 0,C 180,E1 -29355.002,E2 -29355.002} C_VEL
LIN {X 0,Y 127.28,Z 519.727,A -85,B 0,C 180,E1 -29354.768,E2 -29354.768} C_VEL
LIN {X 0,Y 124.662,Z 528.783,A -85,B 0,C 180,E1 -29353.842,E2 -29353.842} C_VEL
LIN {X 0,Y 123.9,Z 531.356,A -85,B 0,C 180,E1 -29353.848,E2 -29353.848} C_VEL
LIN {X 0,Y 119.722,Z 544.143,A -85,B 0,C 180,E1 -29354.629,E2 -29354.629} C_VEL
LIN {X 0,Y 114.917,Z 555.093,A -85,B 0,C 180,E1 -29355.588,E2 -29355.588} C_VEL
LIN {X 0,Y 108.431,Z 566.703,A -85,B 0,C 180,E1 -29357.055,E2 -29357.055} C_VEL
LIN {X 0,Y 101.183,Z 577.138,A -85,B 0,C 180,E1 -29358.85,E2 -29358.85} C_VEL
LIN {X 0,Y 94.051,Z 585.664,A -85,B 0,C 180,E1 -29360.923,E2 -29360.923} C_VEL
LIN {X 0,Y 86.306,Z 593.52,A -85,B 0,C 180,E1 -29363.638,E2 -29363.638} C_VEL
LIN {X 0,Y 77.356,Z 601.188,A -85,B 0,C 180,E1 -29367.649,E2 -29367.649} C_VEL
LIN {X 0,Y 67.403,Z 608.236,A -85,B 0,C 180,E1 -29373.475,E2 -29373.475} C_VEL
LIN {X 0,Y 59.514,Z 612.927,A -85,B 0,C 180,E1 -29379.864,E2 -29379.864} C_VEL
LIN {X 0,Y 52.624,Z 616.51,A -85,B 0,C 180,E1 -29388.108,E2 -29388.108} C_VEL
LIN {X 0,Y 48.719,Z 618.358,A -85,B 0,C 180,E1 -29394.76,E2 -29394.76} C_VEL
LIN {X 0,Y 43.144,Z 620.73,A -85,B 0,C 180,E1 -29410.988,E2 -29410.988} C_VEL
LIN {X 0,Y 41.79,Z 621.331,A -85,B 0,C 180,E1 -29420.32,E2 -29420.32} C_VEL
LIN {X 0,Y 41.418,Z 621.552,A -85,B 0,C 180,E1 -29430.002,E2 -29430.002} C_VEL
LIN {X 0,Y 41.79,Z 621.356,A -85,B 0,C 180,E1 -29439.684,E2 -29439.684} C_VEL
LIN {X 0,Y 45.487,Z 619.801,A -85,B 0,C 180,E1 -29457.616,E2 -29457.616} C_VEL
LIN {X 0,Y 48.714,Z 618.439,A -85,B 0,C 180,E1 -29465.248,E2 -29465.248} C_VEL
LIN {X 0,Y 54.74,Z 615.565,A -85,B 0,C 180,E1 -29474.924,E2 -29474.924} C_VEL
LIN {X 0,Y 62.01,Z 611.662,A -85,B 0,C 180,E1 -29482.503,E2 -29482.503} C_VEL
LIN {X 0,Y 70.164,Z 606.624,A -85,B 0,C 180,E1 -29488.368,E2 -29488.368} C_VEL
LIN {X 0,Y 78.803,Z 600.28,A -85,B 0,C 180,E1 -29493.108,E2 -29493.108} C_VEL
LIN {X 0,Y 87.793,Z 592.349,A -85,B 0,C 180,E1 -29497.016,E2 -29497.016} C_VEL
LIN {X 0,Y 95.573,Z 584.258,A -85,B 0,C 180,E1 -29499.652,E2 -29499.652} C_VEL
LIN {X 0,Y 103.551,Z 574.382,A -85,B 0,C 180,E1 -29501.841,E2 -29501.841} C_VEL
LIN {X 0,Y 110.822,Z 563.249,A -85,B 0,C 180,E1 -29503.577,E2 -29503.577} C_VEL
LIN {X 0,Y 117.214,Z 550.892,A -85,B 0,C 180,E1 -29504.903,E2 -29504.903} C_VEL
LIN {X 0,Y 121.917,Z 538.992,A -85,B 0,C 180,E1 -29505.82,E2 -29505.82} C_VEL
LIN {X 0,Y 125.563,Z 525.974,A -85,B 0,C 180,E1 -29506.52,E2 -29506.52} C_VEL
LIN {X 0,Y 127.171,Z 517.614,A -85,B 0,C 180,E1 -29506.904,E2 -29506.904} C_VEL
LIN {X 0,Y 126.085,Z 513.853,A -85,B 0,C 180,E1 -29510.778,E2 -29510.778} C_VEL
LIN {X 0,Y 125.477,Z 511.649,A -85,B 0,C 180,E1 -29513.972,E2 -29513.972} C_VEL
LIN {X 0,Y 125.107,Z 509.285,A -85,B 0,C 180,E1 -29520,E2 -29520} C_VEL
LIN {X 0,Y 125.703,Z 512.429,A -85,B 0,C 180,E1 -29527.025,E2 -29527.025} C_VEL
LIN {X 0,Y 126.584,Z 515.544,A -85,B 0,C 180,E1 -29530.8,E2 -29530.8} C_VEL
LIN {X 0,Y 127.246,Z 517.664,A -85,B 0,C 180,E1 -29532.874,E2 -29532.874} C_VEL
LIN {X 0,Y 124.666,Z 530.486,A -85,B 0,C 180,E1 -29533.366,E2 -29533.366} C_VEL
LIN {X 0,Y 120.886,Z 542.606,A -85,B 0,C 180,E1 -29533.938,E2 -29533.938} C_VEL
LIN {X 0,Y 116.29,Z 553.705,A -85,B 0,C 180,E1 -29534.765,E2 -29534.765} C_VEL
LIN {X 0,Y 110.512,Z 564.659,A -85,B 0,C 180,E1 -29535.869,E2 -29535.869} C_VEL
LIN {X 0,Y 103.144,Z 575.84,A -85,B 0,C 180,E1 -29537.456,E2 -29537.456} C_VEL
LIN {X 0,Y 95.106,Z 585.765,A -85,B 0,C 180,E1 -29539.576,E2 -29539.576} C_VEL
LIN {X 0,Y 87.203,Z 593.905,A -85,B 0,C 180,E1 -29542.052,E2 -29542.052} C_VEL
LIN {X 0,Y 78.051,Z 601.899,A -85,B 0,C 180,E1 -29545.782,E2 -29545.782} C_VEL
LIN {X 0,Y 68.677,Z 608.759,A -85,B 0,C 180,E1 -29551.003,E2 -29551.003} C_VEL
LIN {X 0,Y 61.258,Z 613.398,A -85,B 0,C 180,E1 -29556.571,E2 -29556.571} C_VEL
LIN {X 0,Y 53.961,Z 617.354,A -85,B 0,C 180,E1 -29564.245,E2 -29564.245} C_VEL
LIN {X 0,Y 47.856,Z 620.28,A -85,B 0,C 180,E1 -29574.023,E2 -29574.023} C_VEL
LIN {X 0,Y 42.616,Z 622.673,A -85,B 0,C 180,E1 -29590.74,E2 -29590.74} C_VEL
LIN {X 0,Y 41.448,Z 623.285,A -85,B 0,C 180,E1 -29600.236,E2 -29600.236} C_VEL
LIN {X 0,Y 41.278,Z 623.499,A -85,B 0,C 180,E1 -29609.998,E2 -29609.998} C_VEL
LIN {X 0,Y 41.447,Z 623.265,A -85,B 0,C 180,E1 -29619.761,E2 -29619.761} C_VEL
LIN {X 0,Y 44.79,Z 621.629,A -85,B 0,C 180,E1 -29638.08,E2 -29638.08} C_VEL
LIN {X 0,Y 47.854,Z 620.214,A -85,B 0,C 180,E1 -29645.975,E2 -29645.975} C_VEL
LIN {X 0,Y 53.958,Z 617.261,A -85,B 0,C 180,E1 -29655.754,E2 -29655.754} C_VEL
LIN {X 0,Y 61.253,Z 613.272,A -85,B 0,C 180,E1 -29663.431,E2 -29663.431} C_VEL
LIN {X 0,Y 70.053,Z 607.652,A -85,B 0,C 180,E1 -29669.893,E2 -29669.893} C_VEL
LIN {X 0,Y 78.035,Z 601.682,A -85,B 0,C 180,E1 -29674.239,E2 -29674.239} C_VEL
LIN {X 0,Y 87.196,Z 593.642,A -85,B 0,C 180,E1 -29677.955,E2 -29677.955} C_VEL
LIN {X 0,Y 95.098,Z 585.45,A -85,B 0,C 180,E1 -29680.433,E2 -29680.433} C_VEL
LIN {X 0,Y 103.14,Z 575.457,A -85,B 0,C 180,E1 -29682.545,E2 -29682.545} C_VEL
LIN {X 0,Y 110.494,Z 564.153,A -85,B 0,C 180,E1 -29684.158,E2 -29684.158} C_VEL
LIN {X 0,Y 116.265,Z 553.073,A -85,B 0,C 180,E1 -29685.278,E2 -29685.278} C_VEL
LIN {X 0,Y 121.076,Z 541.337,A -85,B 0,C 180,E1 -29686.042,E2 -29686.042} C_VEL
LIN {X 0,Y 124.8,Z 528.622,A -85,B 0,C 180,E1 -29686.701,E2 -29686.701} C_VEL
LIN {X 0,Y 126.967,Z 517.447,A -85,B 0,C 180,E1 -29687.097,E2 -29687.097} C_VEL
LIN {X 0,Y 125.801,Z 513.468,A -85,B 0,C 180,E1 -29691.163,E2 -29691.163} C_VEL
LIN {X 0,Y 125.223,Z 511.584,A -85,B 0,C 180,E1 -29693.96,E2 -29693.96} C_VEL
LIN {X 0,Y 124.822,Z 508.837,A -85,B 0,C 180,E1 -29700,E2 -29700} C_VEL
LIN {X 0,Y 124.867,Z 510.298,A -85,B 0,C 180,E1 -29703.631,E2 -29703.631} C_VEL
LIN {X 0,Y 125.455,Z 512.295,A -85,B 0,C 180,E1 -29707.646,E2 -29707.646} C_VEL
LIN {X 0,Y 126.295,Z 515.268,A -85,B 0,C 180,E1 -29711.231,E2 -29711.231} C_VEL
LIN {X 0,Y 126.9,Z 517.365,A -85,B 0,C 180,E1 -29713.206,E2 -29713.206} C_VEL
LIN {X 0,Y 124.448,Z 529.302,A -85,B 0,C 180,E1 -29713.729,E2 -29713.729} C_VEL
LIN {X 0,Y 123.9,Z 531.356,A -85,B 0,C 180,E1 -29713.848,E2 -29713.848} C_VEL
LIN {X 0,Y 122.049,Z 537.01,A -85,B 0,C 180,E1 -29713.783,E2 -29713.783} C_VEL
LIN {X 0,Y 118.112,Z 546.044,A -85,B 0,C 180,E1 -29713.06,E2 -29713.06} C_VEL
LIN {X 0,Y 113.626,Z 554.745,A -85,B 0,C 180,E1 -29712.438,E2 -29712.438} C_VEL
LIN {X 0,Y 110.81,Z 559.83,A -85,B 0,C 180,E1 -29712.604,E2 -29712.604} C_VEL
LIN {X 0,Y 104.067,Z 570.616,A -85,B 0,C 180,E1 -29713.883,E2 -29713.883} C_VEL
LIN {X 0,Y 96.653,Z 580.314,A -85,B 0,C 180,E1 -29715.539,E2 -29715.539} C_VEL
LIN {X 0,Y 88.511,Z 589.14,A -85,B 0,C 180,E1 -29717.669,E2 -29717.669} C_VEL
LIN {X 0,Y 79.793,Z 597.086,A -85,B 0,C 180,E1 -29720.629,E2 -29720.629} C_VEL
LIN {X 0,Y 69.746,Z 604.6,A -85,B 0,C 180,E1 -29724.924,E2 -29724.924} C_VEL
LIN {X 0,Y 60.846,Z 610.094,A -85,B 0,C 180,E1 -29729.972,E2 -29729.972} C_VEL
LIN {X 0,Y 52.527,Z 614.403,A -85,B 0,C 180,E1 -29736.605,E2 -29736.605} C_VEL
LIN {X 0,Y 47.566,Z 616.678,A -85,B 0,C 180,E1 -29742.375,E2 -29742.375} C_VEL
LIN {X 0,Y 43.121,Z 618.526,A -85,B 0,C 180,E1 -29749.315,E2 -29749.315} C_VEL
LIN {X 0,Y 36.496,Z 620.897,A -85,B 0,C 180,E1 -29767.35,E2 -29767.35} C_VEL
LIN {X 0,Y 34.806,Z 621.499,A -85,B 0,C 180,E1 -29778.353,E2 -29778.353} C_VEL
LIN {X 0,Y 34.322,Z 621.719,A -85,B 0,C 180,E1 -29790.002,E2 -29790.002} C_VEL
LIN {X 0,Y 34.807,Z 621.523,A -85,B 0,C 180,E1 -29801.651,E2 -29801.651} C_VEL
LIN {X 0,Y 39.328,Z 619.967,A -85,B 0,C 180,E1 -29822.422,E2 -29822.422} C_VEL
LIN {X 0,Y 43.115,Z 618.605,A -85,B 0,C 180,E1 -29830.697,E2 -29830.697} C_VEL
LIN {X 0,Y 49.957,Z 615.731,A -85,B 0,C 180,E1 -29840.694,E2 -29840.694} C_VEL
LIN {X 0,Y 57.968,Z 611.828,A -85,B 0,C 180,E1 -29848.071,E2 -29848.071} C_VEL
LIN {X 0,Y 66.715,Z 606.79,A -85,B 0,C 180,E1 -29853.566,E2 -29853.566} C_VEL
LIN {X 0,Y 75.86,Z 600.445,A -85,B 0,C 180,E1 -29857.891,E2 -29857.891} C_VEL
LIN {X 0,Y 85.265,Z 592.514,A -85,B 0,C 180,E1 -29861.426,E2 -29861.426} C_VEL
LIN {X 0,Y 93.347,Z 584.422,A -85,B 0,C 180,E1 -29863.73,E2 -29863.73} C_VEL
LIN {X 0,Y 101.562,Z 574.546,A -85,B 0,C 180,E1 -29865.651,E2 -29865.651} C_VEL
LIN {X 0,Y 109.032,Z 563.411,A -85,B 0,C 180,E1 -29867.148,E2 -29867.148} C_VEL
LIN {X 0,Y 115.507,Z 551.186,A -85,B 0,C 180,E1 -29868.289,E2 -29868.289} C_VEL
LIN {X 0,Y 120.563,Z 538.577,A -85,B 0,C 180,E1 -29869.128,E2 -29869.128} C_VEL
LIN {X 0,Y 124.293,Z 525.261,A -85,B 0,C 180,E1 -29869.756,E2 -29869.756} C_VEL
LIN {X 0,Y 124.956,Z 522.059,A -85,B 0,C 180,E1 -29869.944,E2 -29869.944} C_VEL
LIN {X 0,Y 124.372,Z 518.719,A -85,B 0,C 180,E1 -29874.121,E2 -29874.121} C_VEL
LIN {X 0,Y 124.136,Z 516.46,A -85,B 0,C 180,E1 -29880,E2 -29880} C_VEL
LIN {X 0,Y 124.448,Z 519.117,A -85,B 0,C 180,E1 -29886.078,E2 -29886.078} C_VEL
LIN {X 0,Y 125.031,Z 522.142,A -85,B 0,C 180,E1 -29889.82,E2 -29889.82} C_VEL
LIN {X 0,Y 122.063,Z 534.431,A -85,B 0,C 180,E1 -29890.272,E2 -29890.272} C_VEL
LIN {X 0,Y 117.896,Z 546.33,A -85,B 0,C 180,E1 -29890.862,E2 -29890.862} C_VEL
LIN {X 0,Y 112.161,Z 558.549,A -85,B 0,C 180,E1 -29891.74,E2 -29891.74} C_VEL
LIN {X 0,Y 105.418,Z 569.792,A -85,B 0,C 180,E1 -29892.829,E2 -29892.829} C_VEL
LIN {X 0,Y 97.913,Z 579.917,A -85,B 0,C 180,E1 -29894.299,E2 -29894.299} C_VEL
LIN {X 0,Y 89.676,Z 589.048,A -85,B 0,C 180,E1 -29896.248,E2 -29896.248} C_VEL
LIN {X 0,Y 79.968,Z 597.952,A -85,B 0,C 180,E1 -29899.128,E2 -29899.128} C_VEL
LIN {X 0,Y 70.575,Z 605.117,A -85,B 0,C 180,E1 -29902.905,E2 -29902.905} C_VEL
LIN {X 0,Y 60.189,Z 611.649,A -85,B 0,C 180,E1 -29908.864,E2 -29908.864} C_VEL
LIN {X 0,Y 51.85,Z 615.969,A -85,B 0,C 180,E1 -29915.58,E2 -29915.58} C_VEL
LIN {X 0,Y 46.79,Z 618.259,A -85,B 0,C 180,E1 -29921.319,E2 -29921.319} C_VEL
LIN {X 0,Y 42.289,Z 620.113,A -85,B 0,C 180,E1 -29928.333,E2 -29928.333} C_VEL
LIN {X 0,Y 35.976,Z 622.506,A -85,B 0,C 180,E1 -29946.999,E2 -29946.999} C_VEL
LIN {X 0,Y 34.47,Z 623.118,A -85,B 0,C 180,E1 -29958.233,E2 -29958.233} C_VEL
LIN {X 0,Y 34.167,Z 623.332,A -85,B 0,C 180,E1 -29969.998,E2 -29969.998} C_VEL
LIN {X 0,Y 34.47,Z 623.097,A -85,B 0,C 180,E1 -29981.762,E2 -29981.762} C_VEL
LIN {X 0,Y 38.647,Z 621.461,A -85,B 0,C 180,E1 -30003.061,E2 -30003.061} C_VEL
LIN {X 0,Y 42.286,Z 620.045,A -85,B 0,C 180,E1 -30011.665,E2 -30011.665} C_VEL
LIN {X 0,Y 49.25,Z 617.093,A -85,B 0,C 180,E1 -30021.705,E2 -30021.705} C_VEL
LIN {X 0,Y 57.301,Z 613.103,A -85,B 0,C 180,E1 -30029.153,E2 -30029.153} C_VEL
LIN {X 0,Y 66.059,Z 607.949,A -85,B 0,C 180,E1 -30034.814,E2 -30034.814} C_VEL
LIN {X 0,Y 75.212,Z 601.513,A -85,B 0,C 180,E1 -30039.134,E2 -30039.134} C_VEL
LIN {X 0,Y 84.783,Z 593.472,A -85,B 0,C 180,E1 -30042.416,E2 -30042.416} C_VEL
LIN {X 0,Y 92.953,Z 585.279,A -85,B 0,C 180,E1 -30044.579,E2 -30044.579} C_VEL
LIN {X 0,Y 101.236,Z 575.286,A -85,B 0,C 180,E1 -30046.384,E2 -30046.384} C_VEL
LIN {X 0,Y 108.77,Z 563.981,A -85,B 0,C 180,E1 -30047.761,E2 -30047.761} C_VEL
LIN {X 0,Y 114.663,Z 552.9,A -85,B 0,C 180,E1 -30048.719,E2 -30048.719} C_VEL
LIN {X 0,Y 119.877,Z 540.288,A -85,B 0,C 180,E1 -30049.396,E2 -30049.396} C_VEL
LIN {X 0,Y 123.592,Z 527.456,A -85,B 0,C 180,E1 -30049.936,E2 -30049.936} C_VEL
LIN {X 0,Y 124.764,Z 521.87,A -85,B 0,C 180,E1 -30050.159,E2 -30050.159} C_VEL
LIN {X 0,Y 124.184,Z 518.785,A -85,B 0,C 180,E1 -30053.909,E2 -30053.909} C_VEL
LIN {X 0,Y 123.854,Z 516.067,A -85,B 0,C 180,E1 -30060,E2 -30060} C_VEL
LIN {X 0,Y 124.145,Z 518.793,A -85,B 0,C 180,E1 -30066.501,E2 -30066.501} C_VEL
LIN {X 0,Y 124.695,Z 521.899,A -85,B 0,C 180,E1 -30070.243,E2 -30070.243} C_VEL
LIN {X 0,Y 121.602,Z 534.324,A -85,B 0,C 180,E1 -30070.731,E2 -30070.731} C_VEL
LIN {X 0,Y 117.229,Z 546.483,A -85,B 0,C 180,E1 -30071.439,E2 -30071.439} C_VEL
LIN {X 0,Y 111.564,Z 558.422,A -85,B 0,C 180,E1 -30072.468,E2 -30072.468} C_VEL
LIN {X 0,Y 110.81,Z 559.83,A -85,B 0,C 180,E1 -30072.604,E2 -30072.604} C_VEL
LIN {X 0,Y 107.776,Z 564.893,A -85,B 0,C 180,E1 -30072.796,E2 -30072.796} C_VEL
LIN {X 0,Y 101.876,Z 572.812,A -85,B 0,C 180,E1 -30072.258,E2 -30072.258} C_VEL
LIN {X 0,Y 95.365,Z 580.239,A -85,B 0,C 180,E1 -30071.767,E2 -30071.767} C_VEL
LIN {X 0,Y 91.356,Z 584.529,A -85,B 0,C 180,E1 -30072.152,E2 -30072.152} C_VEL
LIN {X 0,Y 81.649,Z 593.859,A -85,B 0,C 180,E1 -30074.457,E2 -30074.457} C_VEL
LIN {X 0,Y 71.883,Z 601.525,A -85,B 0,C 180,E1 -30077.591,E2 -30077.591} C_VEL
LIN {X 0,Y 60.746,Z 608.573,A -85,B 0,C 180,E1 -30082.25,E2 -30082.25} C_VEL
LIN {X 0,Y 51.562,Z 613.264,A -85,B 0,C 180,E1 -30087.633,E2 -30087.633} C_VEL
LIN {X 0,Y 43.096,Z 616.847,A -85,B 0,C 180,E1 -30095.377,E2 -30095.377} C_VEL
LIN {X 0,Y 38.016,Z 618.694,A -85,B 0,C 180,E1 -30102.316,E2 -30102.316} C_VEL
LIN {X 0,Y 30.069,Z 621.065,A -85,B 0,C 180,E1 -30122.134,E2 -30122.134} C_VEL
LIN {X 0,Y 27.898,Z 621.666,A -85,B 0,C 180,E1 -30135.412,E2 -30135.412} C_VEL
LIN {X 0,Y 27.241,Z 621.886,A -85,B 0,C 180,E1 -30150.003,E2 -30150.003} C_VEL
LIN {X 0,Y 27.898,Z 621.689,A -85,B 0,C 180,E1 -30164.594,E2 -30164.594} C_VEL
LIN {X 0,Y 33.553,Z 620.134,A -85,B 0,C 180,E1 -30188.934,E2 -30188.934} C_VEL
LIN {X 0,Y 38.01,Z 618.772,A -85,B 0,C 180,E1 -30197.701,E2 -30197.701} C_VEL
LIN {X 0,Y 45.773,Z 615.898,A -85,B 0,C 180,E1 -30207.619,E2 -30207.619} C_VEL
LIN {X 0,Y 54.539,Z 611.994,A -85,B 0,C 180,E1 -30214.431,E2 -30214.431} C_VEL
LIN {X 0,Y 63.87,Z 606.956,A -85,B 0,C 180,E1 -30219.281,E2 -30219.281} C_VEL
LIN {X 0,Y 73.478,Z 600.61,A -85,B 0,C 180,E1 -30223.039,E2 -30223.039} C_VEL
LIN {X 0,Y 83.277,Z 592.679,A -85,B 0,C 180,E1 -30226.06,E2 -30226.06} C_VEL
LIN {X 0,Y 91.614,Z 584.586,A -85,B 0,C 180,E1 -30227.989,E2 -30227.989} C_VEL
LIN {X 0,Y 100.042,Z 574.709,A -85,B 0,C 180,E1 -30229.587,E2 -30229.587} C_VEL
LIN {X 0,Y 107.679,Z 563.573,A -85,B 0,C 180,E1 -30230.822,E2 -30230.822} C_VEL
LIN {X 0,Y 114.208,Z 551.496,A -85,B 0,C 180,E1 -30231.758,E2 -30231.758} C_VEL
LIN {X 0,Y 119.343,Z 538.995,A -85,B 0,C 180,E1 -30232.461,E2 -30232.461} C_VEL
LIN {X 0,Y 122.885,Z 526.797,A -85,B 0,C 180,E1 -30233.047,E2 -30233.047} C_VEL
LIN {X 0,Y 122.751,Z 525.035,A -85,B 0,C 180,E1 -30235.896,E2 -30235.896} C_VEL
LIN {X 0,Y 122.828,Z 523.573,A -85,B 0,C 180,E1 -30240,E2 -30240} C_VEL
LIN {X 0,Y 122.88,Z 526.03,A -85,B 0,C 180,E1 -30245.538,E2 -30245.538} C_VEL
LIN {X 0,Y 122.965,Z 526.874,A -85,B 0,C 180,E1 -30246.733,E2 -30246.733} C_VEL
LIN {X 0,Y 119.043,Z 540.246,A -85,B 0,C 180,E1 -30247.169,E2 -30247.169} C_VEL
LIN {X 0,Y 114.088,Z 552.196,A -85,B 0,C 180,E1 -30247.773,E2 -30247.773} C_VEL
LIN {X 0,Y 107.5,Z 564.333,A -85,B 0,C 180,E1 -30248.566,E2 -30248.566} C_VEL
LIN {X 0,Y 99.806,Z 575.512,A -85,B 0,C 180,E1 -30249.648,E2 -30249.648} C_VEL
LIN {X 0,Y 91.324,Z 585.435,A -85,B 0,C 180,E1 -30251.12,E2 -30251.12} C_VEL
LIN {X 0,Y 81.245,Z 595.058,A -85,B 0,C 180,E1 -30253.298,E2 -30253.298} C_VEL
LIN {X 0,Y 71.354,Z 602.717,A -85,B 0,C 180,E1 -30256.188,E2 -30256.188} C_VEL
LIN {X 0,Y 60.181,Z 609.793,A -85,B 0,C 180,E1 -30260.89,E2 -30260.89} C_VEL
LIN {X 0,Y 50.974,Z 614.497,A -85,B 0,C 180,E1 -30266.336,E2 -30266.336} C_VEL
LIN {X 0,Y 42.418,Z 618.092,A -85,B 0,C 180,E1 -30274.058,E2 -30274.058} C_VEL
LIN {X 0,Y 37.263,Z 619.945,A -85,B 0,C 180,E1 -30281.021,E2 -30281.021} C_VEL
LIN {X 0,Y 32.911,Z 621.34,A -85,B 0,C 180,E1 -30290.157,E2 -30290.157} C_VEL
LIN {X 0,Y 27.54,Z 622.951,A -85,B 0,C 180,E1 -30315.212,E2 -30315.212} C_VEL
LIN {X 0,Y 27.061,Z 623.165,A -85,B 0,C 180,E1 -30329.997,E2 -30329.997} C_VEL
LIN {X 0,Y 27.539,Z 622.93,A -85,B 0,C 180,E1 -30344.783,E2 -30344.783} C_VEL
LIN {X 0,Y 32.908,Z 621.293,A -85,B 0,C 180,E1 -30369.84,E2 -30369.84} C_VEL
LIN {X 0,Y 37.26,Z 619.877,A -85,B 0,C 180,E1 -30378.978,E2 -30378.978} C_VEL
LIN {X 0,Y 45.183,Z 616.924,A -85,B 0,C 180,E1 -30388.812,E2 -30388.812} C_VEL
LIN {X 0,Y 54.001,Z 612.935,A -85,B 0,C 180,E1 -30395.645,E2 -30395.645} C_VEL
LIN {X 0,Y 63.664,Z 607.579,A -85,B 0,C 180,E1 -30400.841,E2 -30400.841} C_VEL
LIN {X 0,Y 72.982,Z 601.343,A -85,B 0,C 180,E1 -30404.357,E2 -30404.357} C_VEL
